(*
IF bToken THEN
	gUI.TiG.arrPV[1].sColumn[3].bExtend		:=arrExecute[20,0];	//E00L
	gUI.TiG.arrPV[1].sColumn[3].bRetract	:=arrExecute[20,1];	
	gUI.TiG.arrPV[1].sColumn[6].bExtend		:=arrExecute[20,2];	//E01L
	gUI.TiG.arrPV[1].sColumn[6].bRetract	:=arrExecute[20,3];	
	gUI.TiG.arrPV[2].sColumn[1].bExtend		:=arrExecute[20,4];	//E02L
	gUI.TiG.arrPV[2].sColumn[1].bRetract	:=arrExecute[20,5];	
	gUI.TiG.arrPV[2].sColumn[2].bExtend		:=arrExecute[20,6];	//E05L
	gUI.TiG.arrPV[2].sColumn[2].bRetract	:=arrExecute[20,7];	
	gUI.TiG.arrPV[2].sColumn[3].bExtend		:=arrExecute[20,8];	//E06L
	gUI.TiG.arrPV[2].sColumn[3].bRetract	:=arrExecute[20,9];	
	gUI.TiG.arrPV[2].sColumn[4].bExtend		:=arrExecute[20,10];//E09L
	gUI.TiG.arrPV[2].sColumn[4].bRetract	:=arrExecute[20,11];	
	gUI.TiG.arrPV[2].sColumn[5].bExtend		:=arrExecute[20,12];//E10L
	gUI.TiG.arrPV[2].sColumn[5].bRetract	:=arrExecute[20,13];	
	gUI.TiG.arrPV[6].sColumn[4].bExtend		:=arrExecute[20,14];//E13L
	gUI.TiG.arrPV[6].sColumn[4].bRetract	:=arrExecute[20,15];	
			
	gUI.TiG.arrPV[6].sColumn[3].bExtend		:=arrExecute[21,0];	//E14L
	gUI.TiG.arrPV[6].sColumn[3].bRetract	:=arrExecute[21,1];	
	gUI.TiG.arrPV[6].sColumn[5].bExtend		:=arrExecute[21,2];	//E16L1
	gUI.TiG.arrPV[6].sColumn[5].bRetract	:=arrExecute[21,3];	
	gUI.TiG.arrPV[7].sColumn[6].bExtend		:=arrExecute[21,4];	//E17L1
	gUI.TiG.arrPV[7].sColumn[6].bRetract	:=arrExecute[21,5];	
	gUI.TiG.arrPV[7].sColumn[1].bExtend		:=arrExecute[21,6];	//E18L
	gUI.TiG.arrPV[7].sColumn[1].bRetract	:=arrExecute[21,7];	
	gUI.TiG.arrPV[7].sColumn[2].bExtend		:=arrExecute[21,8];	//E22L
	gUI.TiG.arrPV[7].sColumn[2].bRetract	:=arrExecute[21,9];	
	gUI.TiG.arrPV[7].sColumn[3].bExtend		:=arrExecute[21,10];//E23L
	gUI.TiG.arrPV[7].sColumn[3].bRetract	:=arrExecute[21,11];	
	gUI.TiG.arrPV[7].sColumn[7].bExtend		:=arrExecute[21,12];//E27L1
	gUI.TiG.arrPV[7].sColumn[7].bRetract	:=arrExecute[21,13];	
	gUI.TiG.arrPV[1].sColumn[1].bExtend		:=arrExecute[21,14];//E28L1
	gUI.TiG.arrPV[1].sColumn[1].bRetract	:=arrExecute[21,15];	
			
	gUI.TiG.arrPV[1].sColumn[2].bExtend		:=arrExecute[22,0];	//E29L
	gUI.TiG.arrPV[1].sColumn[2].bRetract	:=arrExecute[22,1];	
	gUI.TiG.arrPV[3].sColumn[1].bExtend		:=arrExecute[22,2];	//E01Q1
	gUI.TiG.arrPV[3].sColumn[1].bRetract	:=arrExecute[22,3];	
	gUI.TiG.arrPV[4].sColumn[1].bExtend		:=arrExecute[22,4];	//E05Q1
	gUI.TiG.arrPV[4].sColumn[1].bRetract	:=arrExecute[22,5];	
	gUI.TiG.arrPV[5].sColumn[1].bExtend		:=arrExecute[22,6];	//E09Q1
	gUI.TiG.arrPV[5].sColumn[1].bRetract	:=arrExecute[22,7];	
	gUI.TiG.arrPV[6].sColumn[1].bExtend		:=arrExecute[22,8];	//E13Q
	gUI.TiG.arrPV[6].sColumn[1].bRetract	:=arrExecute[22,9];	
	gUI.TiG.arrPV[6].sColumn[2].bExtend		:=arrExecute[22,10];//E15Q
	gUI.TiG.arrPV[6].sColumn[2].bRetract	:=arrExecute[22,11];	
	gUI.TiG.arrPV[7].sColumn[4].bExtend		:=arrExecute[22,12];//E17Q
	gUI.TiG.arrPV[7].sColumn[4].bRetract	:=arrExecute[22,13];	
	gUI.TiG.arrPV[7].sColumn[5].bExtend		:=arrExecute[22,14];//E22Q
	gUI.TiG.arrPV[7].sColumn[5].bRetract	:=arrExecute[22,15];	
			
	gUI.TiG.arrPV[1].sColumn[5].bExtend		:=arrExecute[23,0];//E28Q
	gUI.TiG.arrPV[1].sColumn[5].bRetract	:=arrExecute[23,1];	
	gUI.TiG.arrPV[1].sColumn[4].bExtend		:=arrExecute[23,2];//E29Q
	gUI.TiG.arrPV[1].sColumn[4].bRetract	:=arrExecute[23,3];	

END_IF

IF bToken THEN
	FOR iTemp1:=20 TO 23 DO
	FOR iTemp2:=0 TO 15 DO
		IF arrExecute[iTemp1,iTemp2] AND isArrived(iTemp1,iTemp2) THEN
			arrExecute[iTemp1,iTemp2]:=0;
		END_IF
	END_FOR		
	END_FOR
END_IF
bToken:=FALSE;
*)
END_METHOD

END_PROGRAM

// Device/Application/public_datum/otherContent/modbusold/isArrived
FUNCTION isArrived : BOOL
VAR_INPUT
	i1		:USINT;
	i2		:USINT;
END_VAR
VAR
	iVT		:USINT;
	iVT1	:USINT;
	i2H	:USINT;	//i2Half
	bFetch	:BOOL;
	
END_VAR
VAR CONSTANT
	a0PV		:ARRAY [0..7] OF USINT :=[1,1,2,2,2,2,2,6];	
	a0PV1		:ARRAY [0..7] OF USINT :=[3,6,1,2,3,4,5,4];		
	a1PV		:ARRAY [0..7] OF USINT :=[6,6,7,7,7,7,7,1];	
	a1PV1		:ARRAY [0..7] OF USINT :=[3,5,6,1,2,3,7,1];	
	a2PV		:ARRAY [0..7] OF USINT :=[1,3,4,5,6,6,7,7];	
	a2PV1		:ARRAY [0..7] OF USINT :=[2,1,1,1,1,2,4,5];		
	a3PV		:ARRAY [0..7] OF USINT :=[1,1];	
	a3PV1		:ARRAY [0..7] OF USINT :=[5,4];	
END_VAR

bFetch:=FALSE;
i2H:=i2/2;
IF i2 MOD 2 =0 THEN//伸出指令
	CASE i1 OF
	20:
		IF gImple.PV_GroupTi.arrPV[a0PV[i2H]].sColumn[a0PV1[i2H]].eStat=cmdStat.Extend_Done THEN
			bFetch:=TRUE;
		END_IF
	21:
		IF gImple.PV_GroupTi.arrPV[a1PV[i2H]].sColumn[a1PV1[i2H]].eStat=cmdStat.Extend_Done THEN
			bFetch:=TRUE;
		END_IF		
	22:
		IF gImple.PV_GroupTi.arrPV[a2PV[i2H]].sColumn[a2PV1[i2H]].eStat=cmdStat.Extend_Done THEN
			bFetch:=TRUE;
		END_IF		
	23:
		IF gImple.PV_GroupTi.arrPV[a2PV[i2H]].sColumn[a2PV1[i2H]].eStat=cmdStat.Extend_Done THEN
			bFetch:=TRUE;
		END_IF		
	END_CASE
ELSE				//缩回指令
		CASE i1 OF
	20:
		IF gImple.PV_GroupTi.arrPV[a0PV[i2H]].sColumn[a0PV1[i2H]].eStat=cmdStat.Retract_Done THEN
			bFetch:=TRUE;
		END_IF
	21:
		IF gImple.PV_GroupTi.arrPV[a1PV[i2H]].sColumn[a1PV1[i2H]].eStat=cmdStat.Retract_Done THEN
			bFetch:=TRUE;
		END_IF		
	22:
		IF gImple.PV_GroupTi.arrPV[a2PV[i2H]].sColumn[a2PV1[i2H]].eStat=cmdStat.Retract_Done THEN
			bFetch:=TRUE;
		END_IF		
	23:
		IF gImple.PV_GroupTi.arrPV[a2PV[i2H]].sColumn[a2PV1[i2H]].eStat=cmdStat.Retract_Done THEN
			bFetch:=TRUE;
		END_IF		
	END_CASE
END_IF


isArrived:=bFetch;

END_FUNCTION

// Device/Application/public_datum/otherContent/rail_rotate/rotatePlatAct
PROGRAM rotatePlatAct
VAR
		bInitialize		:BOOL:=TRUE;
		iTemp			:INT;
		//fbPercentCalc	:percentCalc;
		iV1:INT;
		iV2:INT;
END_VAR

(*
IF bInitialize THEN	//初始化
	rotatePlatAct.initParam();
END_IF
rotatePlatAct.statusDisplayA();
rotatePlatAct.commandDeliverDi();
*)
IF gImple.PV_GroupTi.arrRotSYN.sStatus.oilExtend_Done THEN
	gImple.PV_GroupTi.arrRotSYN.sStatus.oilStat:=cmdStat.Extend_Done;
	gUI.TiG.sRotLed.oilExtended:=TRUE;gUI.TiG.sRotLed.oilRetracted:=FALSE;
END_IF
IF gImple.PV_GroupTi.arrRotSYN.sStatus.oilRetract_Done THEN
	gImple.PV_GroupTi.arrRotSYN.sStatus.oilStat:=cmdStat.Retract_Done;
	gUI.TiG.sRotLed.oilExtended:=FALSE;gUI.TiG.sRotLed.oilRetracted:=TRUE;
END_IF
IF gImple.PV_GroupTi.arrRotSYN.sStatus.rotFront_Done THEN
	gImple.PV_GroupTi.arrRotSYN.sStatus.rotplatformStat:=cmdStat.Extend_Done;
	gUI.TiG.sRotLed.platExtended:=TRUE;gUI.TiG.sRotLed.platRetracted:=FALSE;
END_IF
IF gImple.PV_GroupTi.arrRotSYN.sStatus.rotReverse_Done THEN
	gImple.PV_GroupTi.arrRotSYN.sStatus.rotplatformStat:=cmdStat.Retract_Done;
	gUI.TiG.sRotLed.platExtended:=FALSE;gUI.TiG.sRotLed.platRetracted:=TRUE;
END_IF


	IF gUI.TiG.sRot.oilExtend  THEN
		IF gImple.PV_GroupTi.arrRotSYN.sStatus.oilStat=cmdStat.Extend_Done THEN
			//gImple.PV_GroupTi.arrRotSYN.sStatus.oilCnt:=0;
			gUI.TiG.sRot.oilExtend:=FALSE;
			gImple.PV_GroupTi.arrRotSYN.sCtrl.oilExtend:=FALSE;			
		ELSE
			gImple.PV_GroupTi.arrRotSYN.sStatus.oilStat:=cmdStat.eRun;
			gImple.PV_GroupTi.arrRotSYN.sCtrl.oilExtend:=TRUE;
			gImple.PV_GroupTi.arrRotSYN.sCtrl.oilRetract:=FALSE;
			gUI.TiG.sRot.oilRetract:=FALSE;
		END_IF
	ELSE
		gImple.PV_GroupTi.arrRotSYN.sCtrl.oilExtend:=FALSE;
	END_IF
	
	IF gUI.TiG.sRot.oilRetract  THEN
		IF gImple.PV_GroupTi.arrRotSYN.sStatus.oilStat=cmdStat.Retract_Done THEN
			//gImple.PV_GroupTi.arrRotSYN.sStatus.oilCnt:=0;
			gUI.TiG.sRot.oilRetract:=FALSE;
			gImple.PV_GroupTi.arrRotSYN.sCtrl.oilRetract:=FALSE;
		ELSE
			gImple.PV_GroupTi.arrRotSYN.sStatus.oilStat:=cmdStat.eRun;
			gImple.PV_GroupTi.arrRotSYN.sCtrl.oilRetract:=TRUE;
			gImple.PV_GroupTi.arrRotSYN.sCtrl.oilExtend:=FALSE;	
			gUI.TiG.sRot.oilExtend:=FALSE;	
		END_IF
	ELSE
		gImple.PV_GroupTi.arrRotSYN.sCtrl.oilRetract:=FALSE;
	END_IF	




	IF gUI.TiG.sRot.rotFront  THEN
		IF gImple.PV_GroupTi.arrRotSYN.sStatus.rotplatformStat=cmdStat.Extend_Done THEN
			gUI.TiG.sRot.rotFront:=FALSE;
			gImple.PV_GroupTi.arrRotSYN.sCtrl.rotFront:=FALSE;			
		ELSE 
			gImple.PV_GroupTi.arrRotSYN.sStatus.rotplatformStat:=cmdStat.eRun;
			gImple.PV_GroupTi.arrRotSYN.sCtrl.rotFront:=TRUE;
			gImple.PV_GroupTi.arrRotSYN.sCtrl.rotReverse:=FALSE;	
			gUI.TiG.sRot.rotReverse:=FALSE;
		END_IF
	ELSE
		gImple.PV_GroupTi.arrRotSYN.sCtrl.rotFront:=FALSE;
	END_IF
	
	IF gUI.TiG.sRot.rotReverse  THEN
		IF gImple.PV_GroupTi.arrRotSYN.sStatus.rotplatformStat=cmdStat.Retract_Done THEN
			gUI.TiG.sRot.rotReverse:=FALSE;
			gImple.PV_GroupTi.arrRotSYN.sCtrl.rotReverse:=FALSE;	
		ELSE
			gImple.PV_GroupTi.arrRotSYN.sStatus.rotplatformStat:=cmdStat.eRun;
			gImple.PV_GroupTi.arrRotSYN.sCtrl.rotReverse:=TRUE;
			gImple.PV_GroupTi.arrRotSYN.sCtrl.rotFront:=FALSE;	
			gUI.TiG.sRot.rotFront:=FALSE;
		END_IF
	ELSE
		gImple.PV_GroupTi.arrRotSYN.sCtrl.rotReverse:=FALSE;	
	END_IF

ACTION initParam:
gUI.DiG.arrSYN[31].sNum[1].strName:='D31Q';
gUI.DiG.arrSYN[31].sNum[2].strName:='D31Q1';
gUI.DiG.arrSYN[31].sNum[3].strName:='D31Q2';

gUI.DiG.arrSYN[32].sNum[1].strName:='D32Q';
gUI.DiG.arrSYN[32].sNum[2].strName:='D32Q1';
gUI.DiG.arrSYN[32].sNum[3].strName:='D32Q2';


gUI.TiG.arrSYN[31].sNum[1].strName:='E31Q';
gUI.TiG.arrSYN[31].sNum[2].strName:='E31Q1';
gUI.TiG.arrSYN[32].sNum[1].strName:='E32Q';
gUI.TiG.arrSYN[32].sNum[2].strName:='E32Q2';


//gImple.PV_GroupDi.arrRotSYN[31].arrNum[1].posVal.Retract:=2;
//gImple.PV_GroupDi.arrRotSYN[31].arrNum[1].posVal.Extend:=200;
END_ACTION

ACTION statusDisplayA:
gUI.DiG.arrSYN[31].sNum[1].rPosition:=gImple.PV_GroupDi.arrRotSYN[31].sNum[1].posVal.Current;
gUI.DiG.arrSYN[31].sNum[2].rPosition:=gImple.PV_GroupDi.arrRotSYN[31].sNum[2].posVal.Current;
gUI.DiG.arrSYN[31].sNum[3].rPosition:=gImple.PV_GroupDi.arrRotSYN[31].sNum[3].posVal.Current;

gUI.TiG.arrSYN[31].sNum[1].rPosition:=gImple.PV_GroupTi.arrRotSYN[31].sNum[1].posVal.Current;
gUI.TiG.arrSYN[31].sNum[2].rPosition:=gImple.PV_GroupTi.arrRotSYN[31].sNum[2].posVal.Current;

FOR iTemp:=1 TO 3 DO
	fbPercentCalc(rInput:=gImple.PV_GroupDi.arrRotSYN[31].sNum[iTemp].posVal.Current,
			rExtend:=gImple.PV_GroupDi.arrRotSYN[31].sNum[iTemp].posVal.Extend,
			rRetract:=gImple.PV_GroupDi.arrRotSYN[31].sNum[iTemp].posVal.Retract,
			rOut=>);
	gUI.DiG.arrSYN[31].sNum[iTemp].rPercent:=fbPercentCalc.rOut;
	fbPercentCalc(rInput:=gImple.PV_GroupDi.arrRotSYN[32].sNum[iTemp].posVal.Current,
			rExtend:=gImple.PV_GroupDi.arrRotSYN[32].sNum[iTemp].posVal.Extend,
			rRetract:=gImple.PV_GroupDi.arrRotSYN[32].sNum[iTemp].posVal.Retract,
			rOut=>);
	gUI.DiG.arrSYN[32].sNum[iTemp].rPercent:=fbPercentCalc.rOut;
END_FOR

FOR iTemp:=1 TO 2 DO
	fbPercentCalc(rInput:=gImple.PV_GroupTi.arrRotSYN[31].sNum[iTemp].posVal.Current,
			rExtend:=gImple.PV_GroupTi.arrRotSYN[31].sNum[iTemp].posVal.Extend,
			rRetract:=gImple.PV_GroupTi.arrRotSYN[31].sNum[iTemp].posVal.Retract,
			rOut=>);
	gUI.TiG.arrSYN[31].sNum[iTemp].rPercent:=fbPercentCalc.rOut;
	fbPercentCalc(rInput:=gImple.PV_GroupTi.arrRotSYN[32].sNum[iTemp].posVal.Current,
			rExtend:=gImple.PV_GroupTi.arrRotSYN[32].sNum[iTemp].posVal.Extend,
			rRetract:=gImple.PV_GroupTi.arrRotSYN[32].sNum[iTemp].posVal.Retract,
			rOut=>);
	gUI.TiG.arrSYN[32].sNum[iTemp].rPercent:=fbPercentCalc.rOut;	
END_FOR
END_ACTION

METHOD PRIVATE commandDeliverDi : BOOL
VAR_INPUT
END_VAR
VAR
		eCommand				:cmdStat;
		iCount					:UINT;	
		iCntErr					:UINT:=200*15;			//超时时间15s
		eUnitIndex				:INT;
		fbCheckGroup				:ARRAY[31..32,1..2] OF syncUnitCheck;
		arrOBUSP				:ARRAY[1..2] OF OilBlockUnit_Status_PosVal;

END_VAR
FOR iV1:=31 TO 32 DO
	FOR iV2:=1 TO 2 DO
		iCount:=gImple.PV_GroupDi.arrRotSYN[iV1].iCntErr[iV2];
		IF gUI.DiG.arrSYN[iV1].sColumn[iV2].bExtend<>gUI.DiG.arrSYN[iV1].sColumn[iV2].bRetract THEN
			gImple.PV_GroupDi.arrRotSYN[iV1].sColumn[iV2].eStat:=cmdStat.eRun;
			IF gUI.DiG.arrSYN[iV1].sColumn[iV2].bExtend THEN
				eCommand:=cmdStat.cExtend;
			END_IF
			IF gUI.DiG.arrSYN[iV1].sColumn[iV2].bRetract THEN
				eCommand:=cmdStat.cRetract;
			END_IF
		ELSE	
			eCommand:=cmdStat.cStop;
		END_IF
		IF gUI.DiG.arrSYN[iV1].sColumn[iV2].bStop THEN
			eCommand:=cmdStat.cStop;
		END_IF
		
		arrOBUSP[1].Current:=gImple.PV_GroupDi.arrRotSYN[iV1].sNum[iV2].posVal.Current;
		arrOBUSP[1].Extend:=gImple.PV_GroupDi.arrRotSYN[iV1].sNum[iV2].posVal.Extend;
		arrOBUSP[1].Retract:=gImple.PV_GroupDi.arrRotSYN[iV1].sNum[iV2].posVal.Retract;
		IF iV2=2 THEN
			arrOBUSP[2].Current:=gImple.PV_GroupDi.arrRotSYN[iV1].sNum[iV2].posVal.Current;
			arrOBUSP[2].Extend:=gImple.PV_GroupDi.arrRotSYN[iV1].sNum[iV2].posVal.Extend;
			arrOBUSP[2].Retract:=gImple.PV_GroupDi.arrRotSYN[iV1].sNum[iV2].posVal.Retract;
		ELSE
			arrOBUSP[2].Current:=0;	arrOBUSP[2].Extend:=0;arrOBUSP[2].Retract:=0;
		END_IF
		
		fbCheckGroup[iV1,iV2](
			arrPosVal:=arrOBUSP,
			cmdAct:=eCommand,
			bFetch	=>);
		
		IF fbCheckGroup[iV1,iV2].bFetch=TRUE THEN
			iCount:=0;
			IF gImple.PV_GroupDi.arrRotSYN[iV1].sColumn[iV2].eStat<>cmdStat.eError THEN
				//正常态油缸指令复位
				gUI.DiG.arrSYN[iV1].sColumn[iV2].bStop:=FALSE;
				gUI.DiG.arrSYN[iV1].sColumn[iV2].bExtend:=FALSE;
				gUI.DiG.arrSYN[iV1].sColumn[iV2].bRetract:=FALSE;	
				//SyncCmdExecuteD(ADR(gImple.PV_GroupTi),iV1,iV2,cmdStat.cStop);
				//判断每个开关阀的总状态（伸出or收回）	
				fbCheckGroup[iV1,iV2](cmdAct:=cmdStat.cExtend,arrPosVal:=arrOBUSP);
				IF fbCheckGroup[iV1,iV2].bFetch=TRUE THEN
					gImple.PV_GroupDi.arrRotSYN[iV1].sColumn[iV2].eStat:=cmdStat.Extend_Done;
				END_IF
				fbCheckGroup[iV1,iV2](cmdAct:=cmdStat.cRetract,arrPosVal:=arrOBUSP);
				IF fbCheckGroup[iV1,iV2].bFetch=TRUE THEN
					gImple.PV_GroupDi.arrRotSYN[iV1].sColumn[iV2].eStat:=cmdStat.Retract_Done;
				END_IF			
				//都不是则为Normal态
				IF gImple.PV_GroupDi.arrRotSYN[iV1].sColumn[iV2].eStat<>cmdStat.Retract_Done AND gImple.PV_GroupDi.arrRotSYN[iV1].sColumn[iV2].eStat<>cmdStat.Extend_Done THEN
					gImple.PV_GroupDi.arrRotSYN[iV1].sColumn[iV2].eStat:=cmdStat.eNormal;
				END_IF
				
			END_IF
		ELSE
			iCount:= iCount +1;
			gImple.PV_GroupDi.arrRotSYN[iV1].sColumn[iV2].eStat:=cmdStat.eRun;
			//SyncCmdExecuteD(ADR(gImple.PV_GroupTi),iV1,iV2,eCommand);
		END_IF
		
		IF iCount>=iCntErr THEN
			//错误态油缸指令复位
			gImple.PV_GroupDi.arrRotSYN[iV1].sColumn[iV2].eStat:=cmdStat.eError;
			gUI.DiG.arrSYN[iV1].sColumn[iV2].bStop:=FALSE;
			gUI.DiG.arrSYN[iV1].sColumn[iV2].bExtend:=FALSE;
			gUI.DiG.arrSYN[iV1].sColumn[iV2].bRetract:=FALSE;	
			//SyncCmdExecuteD(ADR(gImple.PV_GroupTi),iV1,iV2,cmdStat.cStop);
		END_IF		
		gImple.PV_GroupDi.arrRotSYN[iV1].iCntErr[iV2]:=iCount;
	END_FOR
END_FOR
END_METHOD

METHOD PRIVATE commandDeliverTi : BOOL
VAR_INPUT
END_VAR
VAR
		eCommand				:cmdStat;
		iCount					:UINT;	
		iCntErr					:UINT:=200*15;			//超时时间15s
		eUnitIndex				:INT;
		fbCheckGroup				:ARRAY[31..32,1..2] OF syncUnitCheck;
		arrOBUSP				:ARRAY[1..2] OF OilBlockUnit_Status_PosVal;

END_VAR
FOR iV1:=31 TO 32 DO
	FOR iV2:=1 TO 2 DO
		iCount:=gImple.PV_GroupTi.arrRotSYN[iV1].iCntErr[iV2];
		IF gUI.TiG.arrSYN[iV1].sColumn[iV2].bExtend<>gUI.TiG.arrSYN[iV1].sColumn[iV2].bRetract THEN
			gImple.PV_GroupTi.arrRotSYN[iV1].sColumn[iV2].eStat:=cmdStat.eRun;
			IF gUI.TiG.arrSYN[iV1].sColumn[iV2].bExtend THEN
				eCommand:=cmdStat.cExtend;
			END_IF
			IF gUI.TiG.arrSYN[iV1].sColumn[iV2].bRetract THEN
				eCommand:=cmdStat.cRetract;
			END_IF
		ELSE	
			eCommand:=cmdStat.cStop;
		END_IF
		IF gUI.TiG.arrSYN[iV1].sColumn[iV2].bStop THEN
			eCommand:=cmdStat.cStop;
		END_IF
		
		arrOBUSP[1].Current:=gImple.PV_GroupTi.arrRotSYN[iV1].sNum[iV2].posVal.Current;
		arrOBUSP[1].Extend:=gImple.PV_GroupTi.arrRotSYN[iV1].sNum[iV2].posVal.Extend;
		arrOBUSP[1].Retract:=gImple.PV_GroupTi.arrRotSYN[iV1].sNum[iV2].posVal.Retract;
		arrOBUSP[2].Current:=0;	arrOBUSP[2].Extend:=0;arrOBUSP[2].Retract:=0;

		
		fbCheckGroup[iV1,iV2](
			arrPosVal:=arrOBUSP,
			cmdAct:=eCommand,
			bFetch	=>);
		
		IF fbCheckGroup[iV1,iV2].bFetch=TRUE THEN
			iCount:=0;
			IF gImple.PV_GroupTi.arrRotSYN[iV1].sColumn[iV2].eStat<>cmdStat.eError THEN
				//正常态油缸指令复位
				gUI.TiG.arrSYN[iV1].sColumn[iV2].bStop:=FALSE;
				gUI.TiG.arrSYN[iV1].sColumn[iV2].bExtend:=FALSE;
				gUI.TiG.arrSYN[iV1].sColumn[iV2].bRetract:=FALSE;	
				//SyncCmdExecuteT(ADR(gImple.PV_GroupTi),iV1,iV2,cmdStat.cStop);
				//判断每个开关阀的总状态（伸出or收回）	
				fbCheckGroup[iV1,iV2](cmdAct:=cmdStat.cExtend,arrPosVal:=arrOBUSP);
				IF fbCheckGroup[iV1,iV2].bFetch=TRUE THEN
					gImple.PV_GroupTi.arrRotSYN[iV1].sColumn[iV2].eStat:=cmdStat.Extend_Done;
				END_IF
				fbCheckGroup[iV1,iV2](cmdAct:=cmdStat.cRetract,arrPosVal:=arrOBUSP);
				IF fbCheckGroup[iV1,iV2].bFetch=TRUE THEN
					gImple.PV_GroupTi.arrRotSYN[iV1].sColumn[iV2].eStat:=cmdStat.Retract_Done;
				END_IF			
				//都不是则为Normal态
				IF gImple.PV_GroupTi.arrRotSYN[iV1].sColumn[iV2].eStat<>cmdStat.Retract_Done AND gImple.PV_GroupTi.arrRotSYN[iV1].sColumn[iV2].eStat<>cmdStat.Extend_Done THEN
					gImple.PV_GroupTi.arrRotSYN[iV1].sColumn[iV2].eStat:=cmdStat.eNormal;
				END_IF
				
			END_IF
		ELSE
			iCount:= iCount +1;
			gImple.PV_GroupTi.arrRotSYN[iV1].sColumn[iV2].eStat:=cmdStat.eRun;
			//SyncCmdExecuteT(ADR(gImple.PV_GroupTi),iV1,iV2,eCommand);
		END_IF
		
		IF iCount>=iCntErr THEN
			//错误态油缸指令复位
			gImple.PV_GroupTi.arrRotSYN[iV1].sColumn[iV2].eStat:=cmdStat.eError;
			gUI.TiG.arrSYN[iV1].sColumn[iV2].bStop:=FALSE;
			gUI.TiG.arrSYN[iV1].sColumn[iV2].bExtend:=FALSE;
			gUI.TiG.arrSYN[iV1].sColumn[iV2].bRetract:=FALSE;	
			//SyncCmdExecuteT(ADR(gImple.PV_GroupTi),iV1,iV2,cmdStat.cStop);
		END_IF		
		gImple.PV_GroupTi.arrRotSYN[iV1].iCntErr[iV2]:=iCount;
	END_FOR
END_FOR
END_METHOD

END_PROGRAM

// Device/Application/public_datum/cmdcheck/syncUnitCheck
FUNCTION_BLOCK syncUnitCheck
VAR_INPUT
	arrPosVal	:ARRAY  [1..2] OF OilBlockUnit_Status_PosVal;

	cmdAct		:cmdStat;
	
END_VAR
VAR_OUTPUT
	bFetch		:BOOL;
END_VAR
VAR
	iCheck			:INT;
	iNum			:INT;				//有值的位移传感器值
	outStat			:ARRAY[1..2] OF OilBlockUnit_Status_Loc;
	iTemp			:INT;
	bAllDone		:BOOL;
END_VAR

iNum:=0;
FOR iTemp :=1 TO 2 DO
	IF arrPosVal[iTemp].Extend <> 0 THEN
		iNum:=iNum+1;
	END_IF
END_FOR
FOR iCheck:=1 TO iNum DO
	outStat[iCheck]	:=fGetUnitStat(arrPosVal[iCheck].Extend,arrPosVal[iCheck].Retract,arrPosVal[iCheck].Current,2.0);
END_FOR


bAllDone:=TRUE;

	//有一个未到指令位置则未完成
	CASE cmdAct OF 
		cmdStat.cExtend:
			FOR iCheck:=1 TO iNum DO
				IF outStat[iCheck]<>OilBlockUnit_Status_Loc.eExtended THEN
					bAllDone:=FALSE;
				END_IF
			END_FOR
		cmdStat.cRetract:
			FOR iCheck:=1 TO iNum DO
				IF outStat[iCheck]<>OilBlockUnit_Status_Loc.eRetracted THEN
					bAllDone:=FALSE;
				END_IF
			END_FOR	
		cmdStat.cStop:
			
	END_CASE

IF bAllDone THEN
	bFetch	:= TRUE;
ELSE
	bFetch	:= FALSE;
END_IF

END_FUNCTION_BLOCK

// Device/Application/can/swmc_floor_rail/swmc_C03_Rx
FUNCTION swmc_C03_Rx : BOOL
VAR_INPUT
	CNT				: UINT;
	//psPVDi			: POINTER TO propValveModule_Di;
	psPVTi			: POINTER TO propValveModule_Ti;
END_VAR
VAR
	frame	 	    : Can_baseframe;
	COB_ID			: UINT;
	I				: UINT;
	pos				: WORD;
END_VAR

IF gCan.C3RxMsg.RxCounter <>  gCan.C3RxCounter THEN    //接收到新的数据

	FOR  I := 1 TO  gCan.C3RxMsg.NoOfRxMessages DO
		frame :=CAN_Read_Data_SWMC(3,I);
		COB_ID :=	frame.id;    //获取ID
		CASE COB_ID OF     //根据ID解析协议
	
			//C3-0x330
			16#330:           //接收C3送来的数据

				psPVTi^.arrRotSYN.sStatus.oilExtend_Done := frame.data[1].0;
				psPVTi^.arrRotSYN.sStatus.oilRetract_Done:= frame.data[1].1;
				
				psPVTi^.arrRotSYN.sStatus.rotFront_Done  := frame.data[2].0;
				psPVTi^.arrRotSYN.sStatus.rotReverse_Done:= frame.data[2].1;
				
		END_CASE
	END_FOR


	gCan.C3RxCounter := gCan.C3RxMsg.RxCounter ;
END_IF

END_FUNCTION

// Device/Application/can/swmc_floor_rail/swmc_C03_Tx
FUNCTION swmc_C03_Tx : BOOL
VAR_INPUT
	CNT				: UINT;
	
	//psPVDi			: POINTER TO propValveModule_Di;
	psPVTi			: POINTER TO propValveModule_Ti;

END_VAR
VAR
	senddata	: ARRAY[1..8] OF BYTE;
	Send_cnt	: UINT;
END_VAR

//速度控制--待定
Send_cnt :=  CNT MOD 3;

CASE Send_cnt OF
	
	1:
 	//C3-0x430
	senddata[1].0 := psPVTi^.arrRotSYN.sCtrl.oilExtend;
	senddata[1].1 := psPVTi^.arrRotSYN.sCtrl.oilRetract;
	
	senddata[2].0 := psPVTi^.arrRotSYN.sCtrl.rotFront;
	senddata[2].1 := psPVTi^.arrRotSYN.sCtrl.rotReverse;	

	//发送至C3
	CAN_Send_Data_SWMC(3, 16#430,senddata);				//发送ID 0x430到C3

END_CASE

END_FUNCTION

// Device/Application/display/OrigDi/YY_Station_Display
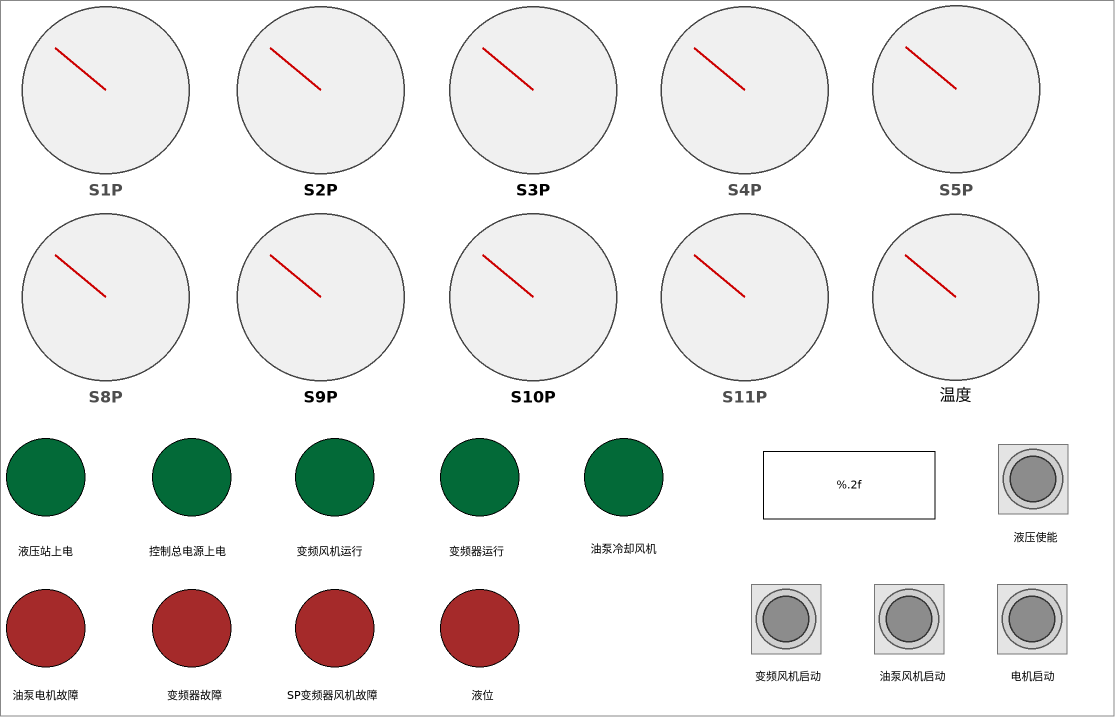
VISUALIZATION YY_Station_Display  // 1115x717
    Ellipse (6,438 79x78), colour toggle: gUI.bYysPower
    Ellipse (152,438 79x78), colour toggle: gUI.bCtrlPower
    Ellipse (295,438 79x78), colour toggle: gUI.bFreqConverterFan
    Ellipse (440,438 79x78), colour toggle: gUI.bFreqConverter
    Label (6,532 79x39), "液压站上电"
    Label (110,532 155x39), "控制总电源上电"
    Label (252,532 155x39), "变频风机运行"
    Label (437,532 79x39), "变频器运行"
    Ellipse (6,589 79x78), colour toggle: gUI.bOilPumpM_Fault
    Ellipse (152,589 79x78), colour toggle: gUI.bFreqConverter_Fault
    Label (6,676 79x39), "油泵电机故障"
    Label (584,532 79x34), "油泵冷却风机"
    Label (117,676 155x39), "变频器故障"
    Ellipse (295,589 79x78), colour toggle: gUI.bFreqConverterFan_Fault
    Label (255,676 155x39), "SP变频器风机故障"
    Ellipse (440,589 79x78), colour toggle: gUI.bFluidLevel
    Label (443,676 79x39), "液位"
    PushSwitchLed (751,584 70x70), variable: gUI.cmdInverterFan, behaviour: TOGGLE, style: Switch-PushSwitchLed-Gray
    PushSwitchLed (874,584 70x70), variable: gUI.cmdOilPumpFan, behaviour: TOGGLE, style: Switch-PushSwitchLed-Gray
    Label (740,657 96x39), "变频风机启动"
    Label (835,657 155x39), "油泵风机启动"
    PushSwitchLed (997,584 70x70), variable: gUI.cmdOilPumpM, behaviour: TOGGLE, style: Switch-PushSwitchLed-Gray
    Label (955,657 155x39), "电机启动"
    Rectangle (763,451 172x68), "%.2f", text variable: gUI.cmdOilPrePercent
        OnMouseDown: write the text variable via Default, min 0, max 100
    Label (958,518 155x39), "液压使能"
    PushSwitchLed (998,444 70x70), variable: gUI.cmdOilPre_EN, behaviour: TOGGLE, style: Switch-PushSwitchLed-Gray
    Ellipse (584,438 79x78), colour toggle: gUI.bOilPumpFan
    Meter360 (872,5 168x168), value: gUI.arrStationPressure[5], style: Meter-Meter360-Gray, scale format: %.1f, scale 0..200
        p518627256: bar
    Label (872,175 168x30), "S5P"
    Meter360 (872,213 167x168), value: gUI.rTemperature, style: Meter-Meter360-Gray, scale format: %.1f, scale 0..200
        p518627256: bar
    Label (872,380 167x30), "温度"
    Meter360 (18,6 175x168), value: gUI.arrStationPressure[1], style: Meter-Meter360-Gray, scale format: %.1f, scale 0..100
        p518627256: bar
    Label (18,175 175x30), "S1P"
    Meter360 (18,213 175x168), value: gUI.arrStationPressure[8], style: Meter-Meter360-Gray, scale format: %.1f, scale 0..100
        p518627256: bar
    Label (18,382 175x30), "S8P"
    Meter360 (234,6 173x168), value: gUI.arrStationPressure[2], style: Meter-Meter360-Gray, scale format: %.1f, scale 0..100
        p518627256: bar
    Label (234,175 173x30), "S2P"
    Meter360 (234,213 173x168), value: gUI.arrStationPressure[9], style: Meter-Meter360-Gray, scale format: %.1f, scale 0..100
        p518627256: bar
    Label (234,382 173x30), "S9P"
    Meter360 (448,6 170x168), value: gUI.arrStationPressure[3], style: Meter-Meter360-Gray, scale format: %.1f, scale 0..100
        p518627256: bar
    Label (448,175 170x30), "S3P"
    Meter360 (448,213 170x168), value: gUI.arrStationPressure[10], style: Meter-Meter360-Gray, scale format: %.1f, scale 0..100
        p518627256: bar
    Label (448,382 170x30), "S10P"
    Meter360 (659,6 171x168), value: gUI.arrStationPressure[4], style: Meter-Meter360-Gray, scale format: %.1f, scale 0..100
        p518627256: bar
    Label (659,175 171x30), "S4P"
    Meter360 (659,213 171x168), value: gUI.arrStationPressure[11], style: Meter-Meter360-Gray, scale format: %.1f, scale 0..100
        p518627256: bar
    Label (659,382 171x30), "S11P"
END_VISUALIZATION

// Device/Application/display/Module/OilBlock_PrimButton
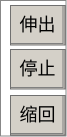
VISUALIZATION OilBlock_PrimButton  // 67x137
VAR_IN_OUT
	extendButton		: BOOL;
	retractButton		: BOOL;
	stopButton			: BOOL;
	
END_VAR
    Button (10,95 55x40), "缩回"
        toggle retractButton
    Button (10,49 55x40), "停止"
        toggle stopButton
    Button (10,5 55x40), "伸出"
        toggle extendButton
END_VISUALIZATION

// Device/Application/display/Module/OilBlock_PrimInfo
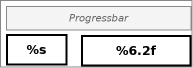
VISUALIZATION OilBlock_PrimInfo  // 193x68
VAR_IN_OUT
	nameStr		:STRING;
	posVal		:REAL;
	percentBar	:REAL;
END_VAR
    RoundedRectangle (6,34 61x31), "%s", text variable: nameStr
    RoundedRectangle (81,35 110x31), "%6.2f", text variable: posVal
    Progressbar (6,6 185x24), variable: percentBar
END_VISUALIZATION

// Device/Application/display/Module/old/Floor_Rail1o
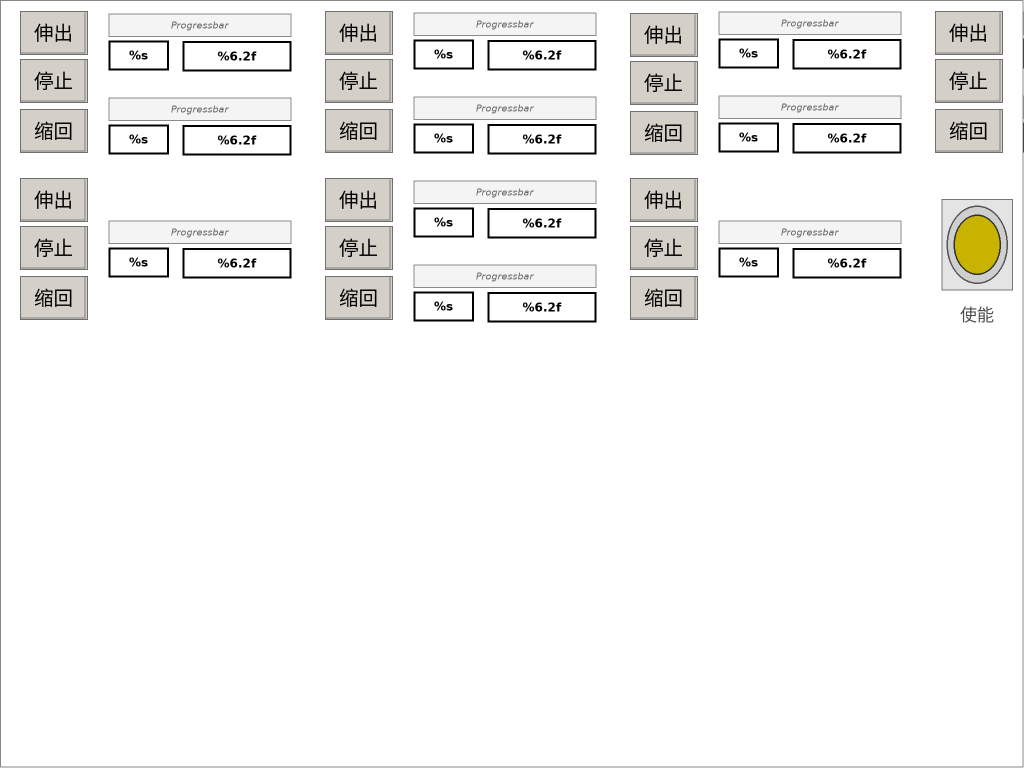
VISUALIZATION Floor_Rail1o  // 1024x768
    Group (8,6 285x151)
        Frame (0,0 82x149)
            shows OilBlock_PrimButton(extendButton := gUI.DiG1.S1.bExtend, retractButton := gUI.DiG1.S1.bRetract, stopButton := gUI.DiG1.S1.bStop)
        Group (95,2 190x149)
            Frame (0,0 190x65)
                shows OilBlock_PrimInfo(nameStr := gUI.DiG1.D00Q1.strName, posVal := gUI.DiG1.D00Q1.rPosition, percentBar := gUI.DiG1.D00Q1.rPercent)
            Frame (0,84 190x65)
                shows OilBlock_PrimInfo(nameStr := gUI.DiG1.D00Q2.strName, posVal := gUI.DiG1.D00Q2.rPosition, percentBar := gUI.DiG1.D00Q2.rPercent)
    Group (313,6 285x150)
        Group (95,1 190x149)
            Frame (0,0 190x65)
                shows OilBlock_PrimInfo(nameStr := gUI.DiG1.D28L1.strName, posVal := gUI.DiG1.D28L1.rPosition, percentBar := gUI.DiG1.D28L1.rPercent)
            Frame (0,84 190x65)
                shows OilBlock_PrimInfo(nameStr := gUI.DiG1.D28L2.strName, posVal := gUI.DiG1.D28L2.rPosition, percentBar := gUI.DiG1.D28L2.rPercent)
        Frame (0,0 82x149)
            shows OilBlock_PrimButton(extendButton := gUI.DiG1.S2.bExtend, retractButton := gUI.DiG1.S2.bRetract, stopButton := gUI.DiG1.S2.bStop)
    Group (618,6 285x151)
        Group (95,0 190x149)
            Frame (0,0 190x65)
                shows OilBlock_PrimInfo(nameStr := gUI.DiG1.D29L.strName, posVal := gUI.DiG1.D29L.rPosition, percentBar := gUI.DiG1.D29L.rPercent)
            Frame (0,84 190x65)
                shows OilBlock_PrimInfo(nameStr := gUI.DiG1.D30L.strName, posVal := gUI.DiG1.D30L.rPosition, percentBar := gUI.DiG1.D30L.rPercent)
        Frame (0,2 82x149)
            shows OilBlock_PrimButton(extendButton := gUI.DiG1.S3.bExtend, retractButton := gUI.DiG1.S3.bRetract, stopButton := gUI.DiG1.S3.bStop)
    Group (923,6 285x149)
        Group (95,0 190x149)
            Frame (0,0 190x65)
                shows OilBlock_PrimInfo(nameStr := gUI.DiG1.D00L1.strName, posVal := gUI.DiG1.D00L1.rPosition, percentBar := gUI.DiG1.D00L1.rPercent)
            Frame (0,84 190x65)
                shows OilBlock_PrimInfo(nameStr := gUI.DiG1.D00L2.strName, posVal := gUI.DiG1.D00L2.rPosition, percentBar := gUI.DiG1.D00L2.rPercent)
        Frame (0,0 82x149)
            shows OilBlock_PrimButton(extendButton := gUI.DiG1.S4.bExtend, retractButton := gUI.DiG1.S4.bRetract, stopButton := gUI.DiG1.S4.bStop)
    Frame (103,215 190x65)
        shows OilBlock_PrimInfo(nameStr := gUI.DiG1.D01L.strName, posVal := gUI.DiG1.D01L.rPosition, percentBar := gUI.DiG1.D01L.rPercent)
    Frame (8,173 82x149)
        shows OilBlock_PrimButton(extendButton := gUI.DiG1.S5.bExtend, retractButton := gUI.DiG1.S5.bRetract, stopButton := gUI.DiG1.S5.bStop)
    Group (313,173 285x151)
        Group (95,2 190x149)
            Frame (0,0 190x65)
                shows OilBlock_PrimInfo(nameStr := gUI.DiG1.D28Q.strName, posVal := gUI.DiG1.D28Q.rPosition, percentBar := gUI.DiG1.D28Q.rPercent)
            Frame (0,84 190x65)
                shows OilBlock_PrimInfo(nameStr := gUI.DiG1.D29Q.strName, posVal := gUI.DiG1.D29Q.rPosition, percentBar := gUI.DiG1.D29Q.rPercent)
        Frame (0,0 82x149)
            shows OilBlock_PrimButton(extendButton := gUI.DiG1.S6.bExtend, retractButton := gUI.DiG1.S6.bRetract, stopButton := gUI.DiG1.S6.bStop)
    Group (618,173 285x149)
        Frame (95,42 190x65)
            shows OilBlock_PrimInfo(nameStr := gUI.DiG1.D30Q.strName, posVal := gUI.DiG1.D30Q.rPosition, percentBar := gUI.DiG1.D30Q.rPercent)
        Frame (0,0 82x149)
            shows OilBlock_PrimButton(extendButton := gUI.DiG1.S7.bExtend, retractButton := gUI.DiG1.S7.bRetract, stopButton := gUI.DiG1.S7.bStop)
    Frame (926,191 285x149)
        shows ModuleDTD(enable := gUI.DiG1.bRVD1_enable, propPercent := gUI.DiG1.rRVD1Percent)
END_VISUALIZATION

// Device/Application/display/Module/ModuleX2
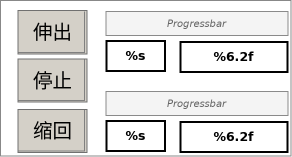
VISUALIZATION ModuleX2  // 292x157
VAR_IN_OUT
	extendButton		: BOOL;
	retractButton		: BOOL;
	stopButton			: BOOL;
	
	nameStr1			:STRING;
	posVal1				:REAL;
	percentBar1			:REAL;
	nameStr2			:STRING;
	posVal2				:REAL;
	percentBar2			:REAL;
END_VAR
    Group (5,5 285x150)
        Frame (0,0 85x150)
            shows OilBlock_PrimButton(extendButton := extendButton, retractButton := retractButton, stopButton := stopButton)
        Frame (95,0 190x70)
            shows OilBlock_PrimInfo(nameStr := nameStr1, posVal := posVal1, percentBar := percentBar1)
        Frame (95,80 190x70)
            shows OilBlock_PrimInfo(nameStr := nameStr2, posVal := posVal2, percentBar := percentBar2)
END_VISUALIZATION

// Device/Application/display/Module/ModuleX1
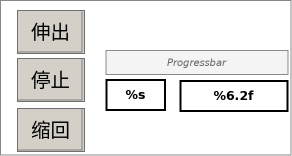
VISUALIZATION ModuleX1  // 292x156
VAR_IN_OUT
	extendButton		: BOOL;
	retractButton		: BOOL;
	stopButton			: BOOL;
	
	nameStr				:STRING;
	posVal				:REAL;
	percentBar			:REAL;
END_VAR
    Group (5,5 285x149)
        Frame (0,0 82x149)
            shows OilBlock_PrimButton(extendButton := extendButton, retractButton := retractButton, stopButton := stopButton)
        Frame (95,39 190x70)
            shows OilBlock_PrimInfo(nameStr := nameStr, posVal := posVal, percentBar := percentBar)
END_VISUALIZATION

// Device/Application/display/Module/ModuleX3
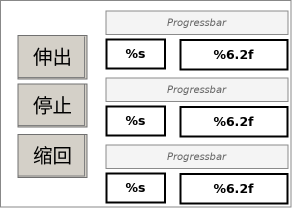
VISUALIZATION ModuleX3  // 292x208
VAR_IN_OUT
	extendButton		: BOOL;
	retractButton		: BOOL;
	stopButton			: BOOL;
	
	nameStr1			:STRING;
	posVal1				:REAL;
	percentBar1			:REAL;
	nameStr2			:STRING;
	posVal2				:REAL;
	percentBar2			:REAL;
	nameStr3			:STRING;
	posVal3				:REAL;
	percentBar3			:REAL;
END_VAR
    Group (5,5 285x201)
        Frame (0,25 85x150)
            shows OilBlock_PrimButton(extendButton := extendButton, retractButton := retractButton, stopButton := stopButton)
        Frame (95,0 190x67)
            shows OilBlock_PrimInfo(nameStr := nameStr1, posVal := posVal1, percentBar := percentBar1)
        Frame (95,67 190x67)
            shows OilBlock_PrimInfo(nameStr := nameStr2, posVal := posVal2, percentBar := percentBar2)
        Frame (95,134 190x67)
            shows OilBlock_PrimInfo(nameStr := nameStr3, posVal := posVal3, percentBar := percentBar3)
END_VISUALIZATION

// Device/Application/display/Module/ModuleX8
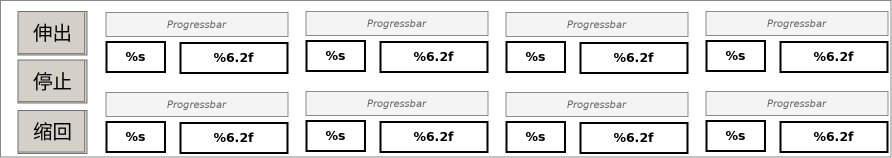
VISUALIZATION ModuleX8  // 892x158
VAR_IN_OUT
	extendButton		: BOOL;
	retractButton		: BOOL;
	stopButton			: BOOL;
	
	nameStr1			:STRING;
	posVal1				:REAL;
	percentBar1			:REAL;
	
	nameStr2			:STRING;
	posVal2				:REAL;
	percentBar2			:REAL;
	
	nameStr3			:STRING;
	posVal3				:REAL;
	percentBar3			:REAL;
	
	nameStr4			:STRING;
	posVal4				:REAL;
	percentBar4			:REAL;
	
	nameStr5			:STRING;
	posVal5				:REAL;
	percentBar5			:REAL;
	
	nameStr6			:STRING;
	posVal6				:REAL;
	percentBar6			:REAL;
	
	nameStr7			:STRING;
	posVal7				:REAL;
	percentBar7			:REAL;
	
	nameStr8			:STRING;
	posVal8				:REAL;
	percentBar8			:REAL;	
	
END_VAR
    Group (5,5 885x151)
        Frame (0,1 85x150)
            shows OilBlock_PrimButton(extendButton := extendButton, retractButton := retractButton, stopButton := stopButton)
        Group (95,0 390x151)
            Group (0,1 190x150)
                Frame (0,0 190x70)
                    shows OilBlock_PrimInfo(nameStr := nameStr1, posVal := posVal1, percentBar := percentBar1)
                Frame (0,80 190x70)
                    shows OilBlock_PrimInfo(nameStr := nameStr2, posVal := posVal2, percentBar := percentBar2)
            Frame (200,0 190x70)
                shows OilBlock_PrimInfo(nameStr := nameStr3, posVal := posVal3, percentBar := percentBar3)
            Frame (200,80 190x70)
                shows OilBlock_PrimInfo(nameStr := nameStr4, posVal := posVal4, percentBar := percentBar4)
        Frame (495,1 190x70)
            shows OilBlock_PrimInfo(nameStr := nameStr5, posVal := posVal5, percentBar := percentBar5)
        Frame (495,81 190x70)
            shows OilBlock_PrimInfo(nameStr := nameStr6, posVal := posVal6, percentBar := percentBar6)
        Frame (695,0 190x70)
            shows OilBlock_PrimInfo(nameStr := nameStr7, posVal := posVal7, percentBar := percentBar7)
        Frame (695,80 190x70)
            shows OilBlock_PrimInfo(nameStr := nameStr8, posVal := posVal8, percentBar := percentBar8)
END_VISUALIZATION

// Device/Application/display/Module/ModuleX4
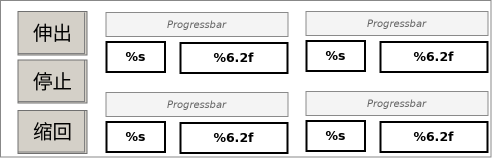
VISUALIZATION ModuleX4  // 492x158
VAR_IN_OUT
	extendButton		: BOOL;
	retractButton		: BOOL;
	stopButton			: BOOL;
	
	nameStr1			:STRING;
	posVal1				:REAL;
	percentBar1			:REAL;
	nameStr2			:STRING;
	posVal2				:REAL;
	percentBar2			:REAL;
	nameStr3			:STRING;
	posVal3				:REAL;
	percentBar3			:REAL;
	nameStr4			:STRING;
	posVal4				:REAL;
	percentBar4			:REAL;
	
	
END_VAR
    Group (5,5 485x151)
        Frame (0,1 85x150)
            shows OilBlock_PrimButton(extendButton := extendButton, retractButton := retractButton, stopButton := stopButton)
        Group (95,1 190x150)
            Frame (0,0 190x70)
                shows OilBlock_PrimInfo(nameStr := nameStr1, posVal := posVal1, percentBar := percentBar1)
            Frame (0,80 190x70)
                shows OilBlock_PrimInfo(nameStr := nameStr2, posVal := posVal2, percentBar := percentBar2)
        Frame (295,0 190x70)
            shows OilBlock_PrimInfo(nameStr := nameStr3, posVal := posVal3, percentBar := percentBar3)
        Frame (295,80 190x70)
            shows OilBlock_PrimInfo(nameStr := nameStr4, posVal := posVal4, percentBar := percentBar4)
END_VISUALIZATION

// Device/Application/display/Module/ModuleX5
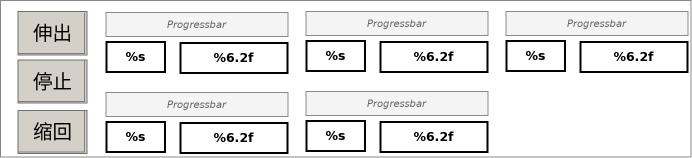
VISUALIZATION ModuleX5  // 692x158
VAR_IN_OUT
	extendButton		: BOOL;
	retractButton		: BOOL;
	stopButton			: BOOL;
	
	nameStr1			:STRING;
	posVal1				:REAL;
	percentBar1			:REAL;
	nameStr2			:STRING;
	posVal2				:REAL;
	percentBar2			:REAL;
	nameStr3			:STRING;
	posVal3				:REAL;
	percentBar3			:REAL;
	nameStr4			:STRING;
	posVal4				:REAL;
	percentBar4			:REAL;
	nameStr5			:STRING;
	posVal5				:REAL;
	percentBar5			:REAL;
	
	
END_VAR
    Group (5,5 685x151)
        Frame (0,1 85x150)
            shows OilBlock_PrimButton(extendButton := extendButton, retractButton := retractButton, stopButton := stopButton)
        Group (95,1 190x150)
            Frame (0,0 190x70)
                shows OilBlock_PrimInfo(nameStr := nameStr1, posVal := posVal1, percentBar := percentBar1)
            Frame (0,80 190x70)
                shows OilBlock_PrimInfo(nameStr := nameStr2, posVal := posVal2, percentBar := percentBar2)
        Frame (295,0 190x70)
            shows OilBlock_PrimInfo(nameStr := nameStr3, posVal := posVal3, percentBar := percentBar3)
        Frame (295,80 190x70)
            shows OilBlock_PrimInfo(nameStr := nameStr4, posVal := posVal4, percentBar := percentBar4)
        Frame (495,0 190x70)
            shows OilBlock_PrimInfo(nameStr := nameStr5, posVal := posVal5, percentBar := percentBar5)
END_VISUALIZATION

// Device/Application/display/OrigTi/Ceiling_Rail2
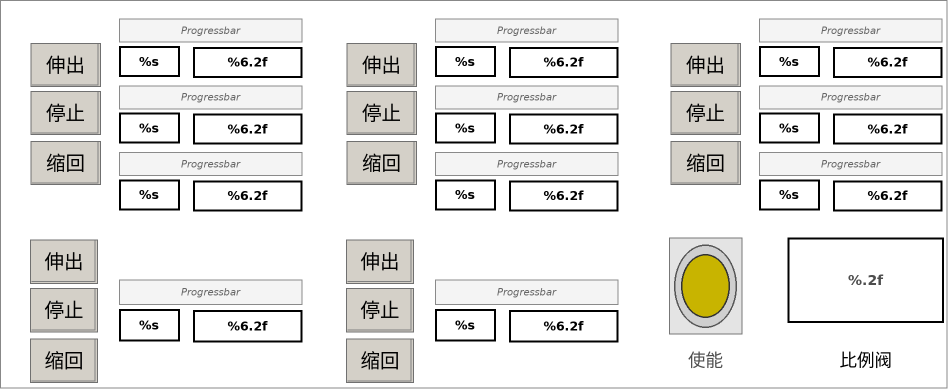
VISUALIZATION Ceiling_Rail2  // 948x389
    Frame (13,8 293x207)
        shows ModuleX3(extendButton := gUI.TiG.arrPV[2].sColumn[1].bExtend, retractButton := gUI.TiG.arrPV[2].sColumn[1].bRetract, stopButton := gUI.TiG.arrPV[2].sColumn[1].bStop, nameStr1 := gUI.TiG.arrPV[2].sNum[1].strName, posVal1 := gUI.TiG.arrPV[2].sNum[1].rPosition, percentBar1 := gUI.TiG.arrPV[2].sNum[1].rPercent, nameStr2 := gUI.TiG.arrPV[2].sNum[2].strName, posVal2 := gUI.TiG.arrPV[2].sNum[2].rPosition, percentBar2 := gUI.TiG.arrPV[2].sNum[2].rPercent, nameStr3 := gUI.TiG.arrPV[2].sNum[3].strName, posVal3 := gUI.TiG.arrPV[2].sNum[3].rPosition, percentBar3 := gUI.TiG.arrPV[2].sNum[3].rPercent)
    Frame (13,229 293x158)
        shows ModuleX1(extendButton := gUI.TiG.arrPV[2].sColumn[2].bExtend, retractButton := gUI.TiG.arrPV[2].sColumn[2].bRetract, stopButton := gUI.TiG.arrPV[2].sColumn[2].bStop, nameStr := gUI.TiG.arrPV[2].sNum[4].strName, posVal := gUI.TiG.arrPV[2].sNum[4].rPosition, percentBar := gUI.TiG.arrPV[2].sNum[4].rPercent)
    Frame (329,8 293x207)
        shows ModuleX3(extendButton := gUI.TiG.arrPV[2].sColumn[3].bExtend, retractButton := gUI.TiG.arrPV[2].sColumn[3].bRetract, stopButton := gUI.TiG.arrPV[2].sColumn[3].bStop, nameStr1 := gUI.TiG.arrPV[2].sNum[5].strName, posVal1 := gUI.TiG.arrPV[2].sNum[5].rPosition, percentBar1 := gUI.TiG.arrPV[2].sNum[5].rPercent, nameStr2 := gUI.TiG.arrPV[2].sNum[6].strName, posVal2 := gUI.TiG.arrPV[2].sNum[6].rPosition, percentBar2 := gUI.TiG.arrPV[2].sNum[6].rPercent, nameStr3 := gUI.TiG.arrPV[2].sNum[7].strName, posVal3 := gUI.TiG.arrPV[2].sNum[7].rPosition, percentBar3 := gUI.TiG.arrPV[2].sNum[7].rPercent)
    Frame (329,229 293x158)
        shows ModuleX1(extendButton := gUI.TiG.arrPV[2].sColumn[4].bExtend, retractButton := gUI.TiG.arrPV[2].sColumn[4].bRetract, stopButton := gUI.TiG.arrPV[2].sColumn[4].bStop, nameStr := gUI.TiG.arrPV[2].sNum[8].strName, posVal := gUI.TiG.arrPV[2].sNum[8].rPosition, percentBar := gUI.TiG.arrPV[2].sNum[8].rPercent)
    Frame (653,8 293x207)
        shows ModuleX3(extendButton := gUI.TiG.arrPV[2].sColumn[5].bExtend, retractButton := gUI.TiG.arrPV[2].sColumn[5].bRetract, stopButton := gUI.TiG.arrPV[2].sColumn[5].bStop, nameStr1 := gUI.TiG.arrPV[2].sNum[9].strName, posVal1 := gUI.TiG.arrPV[2].sNum[9].rPosition, percentBar1 := gUI.TiG.arrPV[2].sNum[9].rPercent, nameStr2 := gUI.TiG.arrPV[2].sNum[10].strName, posVal2 := gUI.TiG.arrPV[2].sNum[10].rPosition, percentBar2 := gUI.TiG.arrPV[2].sNum[10].rPercent, nameStr3 := gUI.TiG.arrPV[2].sNum[11].strName, posVal3 := gUI.TiG.arrPV[2].sNum[11].rPosition, percentBar3 := gUI.TiG.arrPV[2].sNum[11].rPercent)
    Frame (653,229 293x158)
        shows ModuleDTD(enable := gUI.TiG.arrPV[2].bPVD_enable, propPercent := gUI.TiG.arrPV[2].rPVDPercent)
END_VISUALIZATION

// Device/Application/display/Module/ModuleDTD
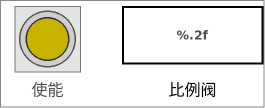
VISUALIZATION ModuleDTD  // 265x108
VAR_IN_OUT
	enable			:BOOL;
	propPercent		:REAL;
END_VAR
    Rectangle (122,6 141x58), "%.2f", text variable: propPercent
        OnMouseDown: write the text variable via Default, min 0, max 100
    Label (122,74 141x32), "比例阀"
    PushSwitchLed (13,6 69x66), variable: enable, behaviour: TOGGLE, style: Switch-PushSwitchLed-Yellow
    Label (13,74 69x32), "使能"
END_VISUALIZATION

// Device/Application/display/OrigDi/Floor_Rail_345
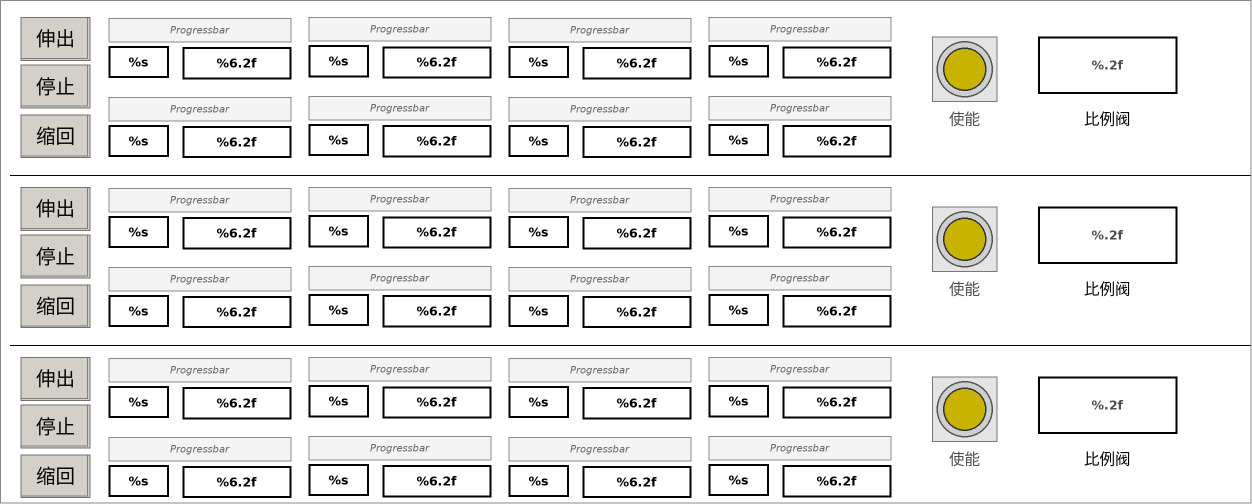
VISUALIZATION Floor_Rail_345  // 1252x504
    Frame (3,6 892x156)
        shows ModuleX8(extendButton := gUI.DiG.arrPV[3].sColumn[1].bExtend, retractButton := gUI.DiG.arrPV[3].sColumn[1].bRetract, stopButton := gUI.DiG.arrPV[3].sColumn[1].bStop, nameStr1 := gUI.DiG.arrPV[3].sNum[1].strName, posVal1 := gUI.DiG.arrPV[3].sNum[1].rPosition, percentBar1 := gUI.DiG.arrPV[3].sNum[1].rPercent, nameStr2 := gUI.DiG.arrPV[3].sNum[2].strName, posVal2 := gUI.DiG.arrPV[3].sNum[2].rPosition, percentBar2 := gUI.DiG.arrPV[3].sNum[2].rPercent, nameStr3 := gUI.DiG.arrPV[3].sNum[3].strName, posVal3 := gUI.DiG.arrPV[3].sNum[3].rPosition, percentBar3 := gUI.DiG.arrPV[3].sNum[3].rPercent, nameStr4 := gUI.DiG.arrPV[3].sNum[4].strName, posVal4 := gUI.DiG.arrPV[3].sNum[4].rPosition, percentBar4 := gUI.DiG.arrPV[3].sNum[4].rPercent, nameStr5 := gUI.DiG.arrPV[3].sNum[5].strName, posVal5 := gUI.DiG.arrPV[3].sNum[5].rPosition, percentBar5 := gUI.DiG.arrPV[3].sNum[5].rPercent, nameStr6 := gUI.DiG.arrPV[3].sNum[6].strName, posVal6 := gUI.DiG.arrPV[3].sNum[6].rPosition, percentBar6 := gUI.DiG.arrPV[3].sNum[6].rPercent, nameStr7 := gUI.DiG.arrPV[3].sNum[7].strName, posVal7 := gUI.DiG.arrPV[3].sNum[7].rPosition, percentBar7 := gUI.DiG.arrPV[3].sNum[7].rPercent, nameStr8 := gUI.DiG.arrPV[3].sNum[8].strName, posVal8 := gUI.DiG.arrPV[3].sNum[8].rPosition, percentBar8 := gUI.DiG.arrPV[3].sNum[8].rPercent)
    Frame (3,176 892x156)
        shows ModuleX8(extendButton := gUI.DiG.arrPV[4].sColumn[1].bExtend, retractButton := gUI.DiG.arrPV[4].sColumn[1].bRetract, stopButton := gUI.DiG.arrPV[4].sColumn[1].bStop, nameStr1 := gUI.DiG.arrPV[4].sNum[1].strName, posVal1 := gUI.DiG.arrPV[4].sNum[1].rPosition, percentBar1 := gUI.DiG.arrPV[4].sNum[1].rPercent, nameStr2 := gUI.DiG.arrPV[4].sNum[2].strName, posVal2 := gUI.DiG.arrPV[4].sNum[2].rPosition, percentBar2 := gUI.DiG.arrPV[4].sNum[2].rPercent, nameStr3 := gUI.DiG.arrPV[4].sNum[3].strName, posVal3 := gUI.DiG.arrPV[4].sNum[3].rPosition, percentBar3 := gUI.DiG.arrPV[4].sNum[3].rPercent, nameStr4 := gUI.DiG.arrPV[4].sNum[4].strName, posVal4 := gUI.DiG.arrPV[4].sNum[4].rPosition, percentBar4 := gUI.DiG.arrPV[4].sNum[4].rPercent, nameStr5 := gUI.DiG.arrPV[4].sNum[5].strName, posVal5 := gUI.DiG.arrPV[4].sNum[5].rPosition, percentBar5 := gUI.DiG.arrPV[4].sNum[5].rPercent, nameStr6 := gUI.DiG.arrPV[4].sNum[6].strName, posVal6 := gUI.DiG.arrPV[4].sNum[6].rPosition, percentBar6 := gUI.DiG.arrPV[4].sNum[6].rPercent, nameStr7 := gUI.DiG.arrPV[4].sNum[7].strName, posVal7 := gUI.DiG.arrPV[4].sNum[7].rPosition, percentBar7 := gUI.DiG.arrPV[4].sNum[7].rPercent, nameStr8 := gUI.DiG.arrPV[4].sNum[8].strName, posVal8 := gUI.DiG.arrPV[4].sNum[8].rPosition, percentBar8 := gUI.DiG.arrPV[4].sNum[8].rPercent)
    Frame (3,346 892x156)
        shows ModuleX8(extendButton := gUI.DiG.arrPV[5].sColumn[1].bExtend, retractButton := gUI.DiG.arrPV[5].sColumn[1].bStop, stopButton := gUI.DiG.arrPV[5].sColumn[1].bStop, nameStr1 := gUI.DiG.arrPV[5].sNum[1].strName, posVal1 := gUI.DiG.arrPV[5].sNum[1].rPosition, percentBar1 := gUI.DiG.arrPV[5].sNum[1].rPercent, nameStr2 := gUI.DiG.arrPV[5].sNum[2].strName, posVal2 := gUI.DiG.arrPV[5].sNum[2].rPosition, percentBar2 := gUI.DiG.arrPV[5].sNum[2].rPercent, nameStr3 := gUI.DiG.arrPV[5].sNum[3].strName, posVal3 := gUI.DiG.arrPV[5].sNum[3].rPosition, percentBar3 := gUI.DiG.arrPV[5].sNum[3].rPercent, nameStr4 := gUI.DiG.arrPV[5].sNum[4].strName, posVal4 := gUI.DiG.arrPV[5].sNum[4].rPosition, percentBar4 := gUI.DiG.arrPV[5].sNum[4].rPercent, nameStr5 := gUI.DiG.arrPV[5].sNum[5].strName, posVal5 := gUI.DiG.arrPV[5].sNum[5].rPosition, percentBar5 := gUI.DiG.arrPV[5].sNum[5].rPercent, nameStr6 := gUI.DiG.arrPV[5].sNum[6].strName, posVal6 := gUI.DiG.arrPV[5].sNum[6].rPosition, percentBar6 := gUI.DiG.arrPV[5].sNum[6].rPercent, nameStr7 := gUI.DiG.arrPV[5].sNum[7].strName, posVal7 := gUI.DiG.arrPV[5].sNum[7].rPosition, percentBar7 := gUI.DiG.arrPV[5].sNum[7].rPercent, nameStr8 := gUI.DiG.arrPV[5].sNum[8].strName, posVal8 := gUI.DiG.arrPV[5].sNum[8].rPosition, percentBar8 := gUI.DiG.arrPV[5].sNum[8].rPercent)
    Frame (918,31 261x106)
        shows ModuleDTD(enable := gUI.DiG.arrPV[3].bPVD_enable, propPercent := gUI.DiG.arrPV[3].rPVDPercent)
    Frame (918,201 261x106)
        shows ModuleDTD(enable := gUI.DiG.arrPV[4].bPVD_enable, propPercent := gUI.DiG.arrPV[4].rPVDPercent)
    Frame (918,371 261x106)
        shows ModuleDTD(enable := gUI.DiG.arrPV[5].bPVD_enable, propPercent := gUI.DiG.arrPV[5].rPVDPercent)
    Line (10,175) (1250,175)
    Line (10,345) (1250,345)
END_VISUALIZATION

// Device/Application/display/OrigDi/Floor_Rail6
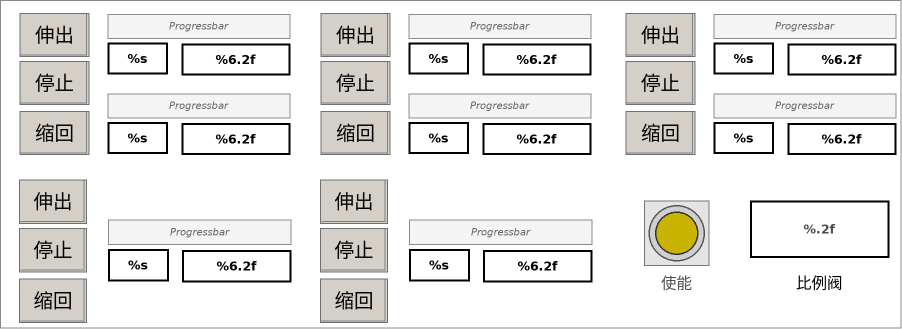
VISUALIZATION Floor_Rail6  // 902x329
    Frame (2,169 293x158)
        shows ModuleX1(extendButton := gUI.DiG.arrPV[6].sColumn[2].bExtend, retractButton := gUI.DiG.arrPV[6].sColumn[2].bRetract, stopButton := gUI.DiG.arrPV[6].sColumn[2].bStop, nameStr := gUI.DiG.arrPV[6].sNum[3].strName, posVal := gUI.DiG.arrPV[6].sNum[3].rPosition, percentBar := gUI.DiG.arrPV[6].sNum[3].rPercent)
    Frame (2,3 292x156)
        shows ModuleX2(extendButton := gUI.DiG.arrPV[6].sColumn[1].bExtend, retractButton := gUI.DiG.arrPV[6].sColumn[1].bRetract, stopButton := gUI.DiG.arrPV[6].sColumn[1].bStop, nameStr1 := gUI.DiG.arrPV[6].sNum[1].strName, posVal1 := gUI.DiG.arrPV[6].sNum[1].rPosition, percentBar1 := gUI.DiG.arrPV[6].sNum[1].rPercent, nameStr2 := gUI.DiG.arrPV[6].sNum[2].strName, posVal2 := gUI.DiG.arrPV[6].sNum[2].rPosition, percentBar2 := gUI.DiG.arrPV[6].sNum[2].rPercent)
    Frame (303,3 292x156)
        shows ModuleX2(extendButton := gUI.DiG.arrPV[6].sColumn[3].bExtend, retractButton := gUI.DiG.arrPV[6].sColumn[3].bRetract, stopButton := gUI.DiG.arrPV[6].sColumn[3].bStop, nameStr1 := gUI.DiG.arrPV[6].sNum[4].strName, posVal1 := gUI.DiG.arrPV[6].sNum[4].rPosition, percentBar1 := gUI.DiG.arrPV[6].sNum[4].rPercent, nameStr2 := gUI.DiG.arrPV[6].sNum[5].strName, posVal2 := gUI.DiG.arrPV[6].sNum[5].rPosition, percentBar2 := gUI.DiG.arrPV[6].sNum[5].rPercent)
    Frame (303,169 293x158)
        shows ModuleX1(extendButton := gUI.DiG.arrPV[6].sColumn[4].bExtend, retractButton := gUI.DiG.arrPV[6].sColumn[4].bRetract, stopButton := gUI.DiG.arrPV[6].sColumn[4].bStop, nameStr := gUI.DiG.arrPV[6].sNum[6].strName, posVal := gUI.DiG.arrPV[6].sNum[6].rPosition, percentBar := gUI.DiG.arrPV[6].sNum[6].rPercent)
    Frame (608,3 292x156)
        shows ModuleX2(extendButton := gUI.DiG.arrPV[6].sColumn[5].bExtend, retractButton := gUI.DiG.arrPV[6].sColumn[5].bRetract, stopButton := gUI.DiG.arrPV[6].sColumn[5].bStop, nameStr1 := gUI.DiG.arrPV[6].sNum[7].strName, posVal1 := gUI.DiG.arrPV[6].sNum[7].rPosition, percentBar1 := gUI.DiG.arrPV[6].sNum[7].rPercent, nameStr2 := gUI.DiG.arrPV[6].sNum[8].strName, posVal2 := gUI.DiG.arrPV[6].sNum[8].rPosition, percentBar2 := gUI.DiG.arrPV[6].sNum[8].rPercent)
    Frame (630,195 261x106)
        shows ModuleDTD(enable := gUI.DiG.arrPV[6].bPVD_enable, propPercent := gUI.DiG.arrPV[6].rPVDPercent)
END_VISUALIZATION

// Device/Application/display/OrigDi/Floor_Rail7
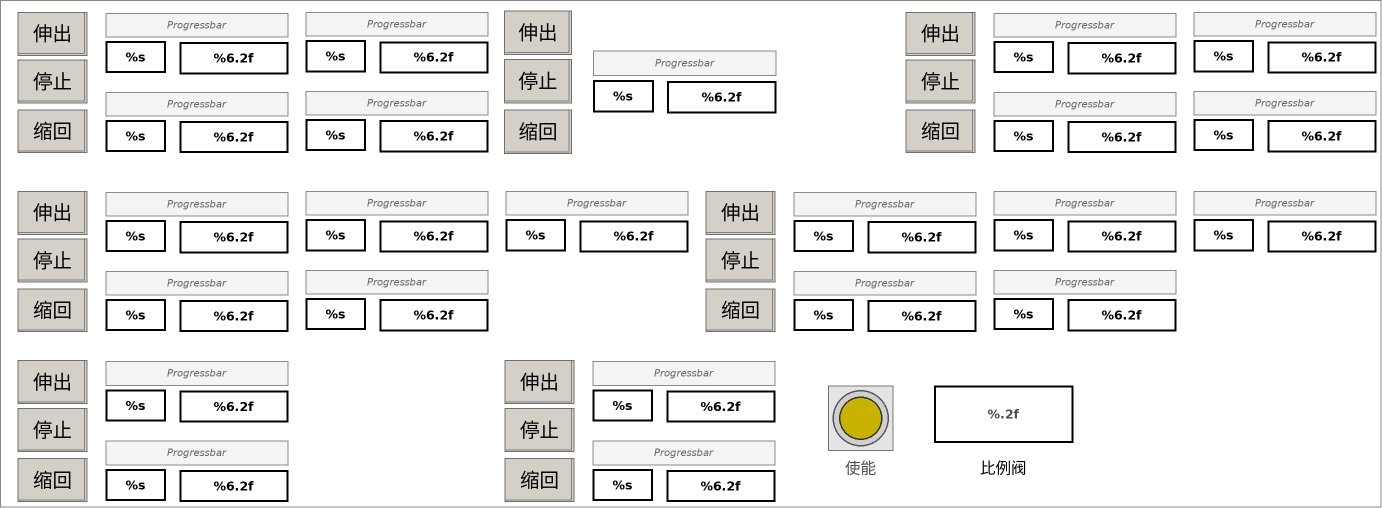
VISUALIZATION Floor_Rail7  // 1382x508
    Frame (0,1 492x156)
        shows ModuleX4(extendButton := gUI.DiG.arrPV[7].sColumn[1].bExtend, retractButton := gUI.DiG.arrPV[7].sColumn[1].bRetract, stopButton := gUI.DiG.arrPV[7].sColumn[1].bStop, nameStr1 := gUI.DiG.arrPV[7].sNum[1].strName, posVal1 := gUI.DiG.arrPV[7].sNum[1].rPosition, percentBar1 := gUI.DiG.arrPV[7].sNum[1].rPercent, nameStr2 := gUI.DiG.arrPV[7].sNum[2].strName, posVal2 := gUI.DiG.arrPV[7].sNum[2].rPosition, percentBar2 := gUI.DiG.arrPV[7].sNum[2].rPercent, nameStr3 := gUI.DiG.arrPV[7].sNum[3].strName, posVal3 := gUI.DiG.arrPV[7].sNum[3].rPosition, percentBar3 := gUI.DiG.arrPV[7].sNum[3].rPercent, nameStr4 := gUI.DiG.arrPV[7].sNum[4].strName, posVal4 := gUI.DiG.arrPV[7].sNum[4].rPosition, percentBar4 := gUI.DiG.arrPV[7].sNum[4].rPercent)
    Frame (487,0 293x158)
        shows ModuleX1(extendButton := gUI.DiG.arrPV[7].sColumn[2].bExtend, retractButton := gUI.DiG.arrPV[7].sColumn[2].bRetract, stopButton := gUI.DiG.arrPV[7].sColumn[2].bStop, nameStr := gUI.DiG.arrPV[7].sNum[5].strName, posVal := gUI.DiG.arrPV[7].sNum[5].rPosition, percentBar := gUI.DiG.arrPV[7].sNum[5].rPercent)
    Frame (888,1 492x156)
        shows ModuleX4(extendButton := gUI.DiG.arrPV[7].sColumn[3].bExtend, retractButton := gUI.DiG.arrPV[7].sColumn[3].bRetract, stopButton := gUI.DiG.arrPV[7].sColumn[3].bStop, nameStr1 := gUI.DiG.arrPV[7].sNum[6].strName, posVal1 := gUI.DiG.arrPV[7].sNum[6].rPosition, percentBar1 := gUI.DiG.arrPV[7].sNum[6].rPercent, nameStr2 := gUI.DiG.arrPV[7].sNum[7].strName, posVal2 := gUI.DiG.arrPV[7].sNum[7].rPosition, percentBar2 := gUI.DiG.arrPV[7].sNum[7].rPercent, nameStr3 := gUI.DiG.arrPV[7].sNum[8].strName, posVal3 := gUI.DiG.arrPV[7].sNum[8].rPosition, percentBar3 := gUI.DiG.arrPV[7].sNum[8].rPercent, nameStr4 := gUI.DiG.arrPV[7].sNum[9].strName, posVal4 := gUI.DiG.arrPV[7].sNum[9].rPosition, percentBar4 := gUI.DiG.arrPV[7].sNum[9].rPercent)
    Frame (0,180 692x156)
        shows ModuleX5(extendButton := gUI.DiG.arrPV[7].sColumn[4].bExtend, retractButton := gUI.DiG.arrPV[7].sColumn[4].bRetract, stopButton := gUI.DiG.arrPV[7].sColumn[4].bStop, nameStr1 := gUI.DiG.arrPV[7].sNum[10].strName, posVal1 := gUI.DiG.arrPV[7].sNum[10].rPosition, percentBar1 := gUI.DiG.arrPV[7].sNum[10].rPercent, nameStr2 := gUI.DiG.arrPV[7].sNum[11].strName, posVal2 := gUI.DiG.arrPV[7].sNum[11].rPosition, percentBar2 := gUI.DiG.arrPV[7].sNum[11].rPercent, nameStr3 := gUI.DiG.arrPV[7].sNum[12].strName, posVal3 := gUI.DiG.arrPV[7].sNum[12].rPosition, percentBar3 := gUI.DiG.arrPV[7].sNum[12].rPercent, nameStr4 := gUI.DiG.arrPV[7].sNum[13].strName, posVal4 := gUI.DiG.arrPV[7].sNum[13].rPosition, percentBar4 := gUI.DiG.arrPV[7].sNum[13].rPercent, nameStr5 := gUI.DiG.arrPV[7].sNum[14].strName, posVal5 := gUI.DiG.arrPV[7].sNum[14].rPosition, percentBar5 := gUI.DiG.arrPV[7].sNum[14].rPercent)
    Frame (688,180 692x156)
        shows ModuleX5(extendButton := gUI.DiG.arrPV[7].sColumn[5].bExtend, retractButton := gUI.DiG.arrPV[7].sColumn[5].bRetract, stopButton := gUI.DiG.arrPV[7].sColumn[5].bStop, nameStr1 := gUI.DiG.arrPV[7].sNum[15].strName, posVal1 := gUI.DiG.arrPV[7].sNum[15].rPosition, percentBar1 := gUI.DiG.arrPV[7].sNum[15].rPercent, nameStr2 := gUI.DiG.arrPV[7].sNum[16].strName, posVal2 := gUI.DiG.arrPV[7].sNum[16].rPosition, percentBar2 := gUI.DiG.arrPV[7].sNum[16].rPercent, nameStr3 := gUI.DiG.arrPV[7].sNum[17].strName, posVal3 := gUI.DiG.arrPV[7].sNum[17].rPosition, percentBar3 := gUI.DiG.arrPV[7].sNum[17].rPercent, nameStr4 := gUI.DiG.arrPV[7].sNum[18].strName, posVal4 := gUI.DiG.arrPV[7].sNum[18].rPosition, percentBar4 := gUI.DiG.arrPV[7].sNum[18].rPercent, nameStr5 := gUI.DiG.arrPV[7].sNum[19].strName, posVal5 := gUI.DiG.arrPV[7].sNum[19].rPosition, percentBar5 := gUI.DiG.arrPV[7].sNum[19].rPercent)
    Frame (0,350 292x156)
        shows ModuleX2(extendButton := gUI.DiG.arrPV[7].sColumn[6].bExtend, retractButton := gUI.DiG.arrPV[7].sColumn[6].bRetract, stopButton := gUI.DiG.arrPV[7].sColumn[6].bStop, nameStr1 := gUI.DiG.arrPV[7].sNum[20].strName, posVal1 := gUI.DiG.arrPV[7].sNum[20].rPosition, percentBar1 := gUI.DiG.arrPV[7].sNum[20].rPercent, nameStr2 := gUI.DiG.arrPV[7].sNum[21].strName, posVal2 := gUI.DiG.arrPV[7].sNum[21].rPosition, percentBar2 := gUI.DiG.arrPV[7].sNum[21].rPercent)
    Frame (487,350 292x156)
        shows ModuleX2(extendButton := gUI.DiG.arrPV[7].sColumn[7].bExtend, retractButton := gUI.DiG.arrPV[7].sColumn[7].bRetract, stopButton := gUI.DiG.arrPV[7].sColumn[7].bStop, nameStr1 := gUI.DiG.arrPV[7].sNum[22].strName, posVal1 := gUI.DiG.arrPV[7].sNum[22].rPosition, percentBar1 := gUI.DiG.arrPV[7].sNum[22].rPercent, nameStr2 := gUI.DiG.arrPV[7].sNum[23].strName, posVal2 := gUI.DiG.arrPV[7].sNum[23].rPosition, percentBar2 := gUI.DiG.arrPV[7].sNum[23].rPercent)
    Frame (814,380 261x106)
        shows ModuleDTD(enable := gUI.DiG.arrPV[7].bPVD_enable, propPercent := gUI.DiG.arrPV[7].rPVDPercent)
END_VISUALIZATION

// Device/Application/display/Module/old/Floor_Rail_12o
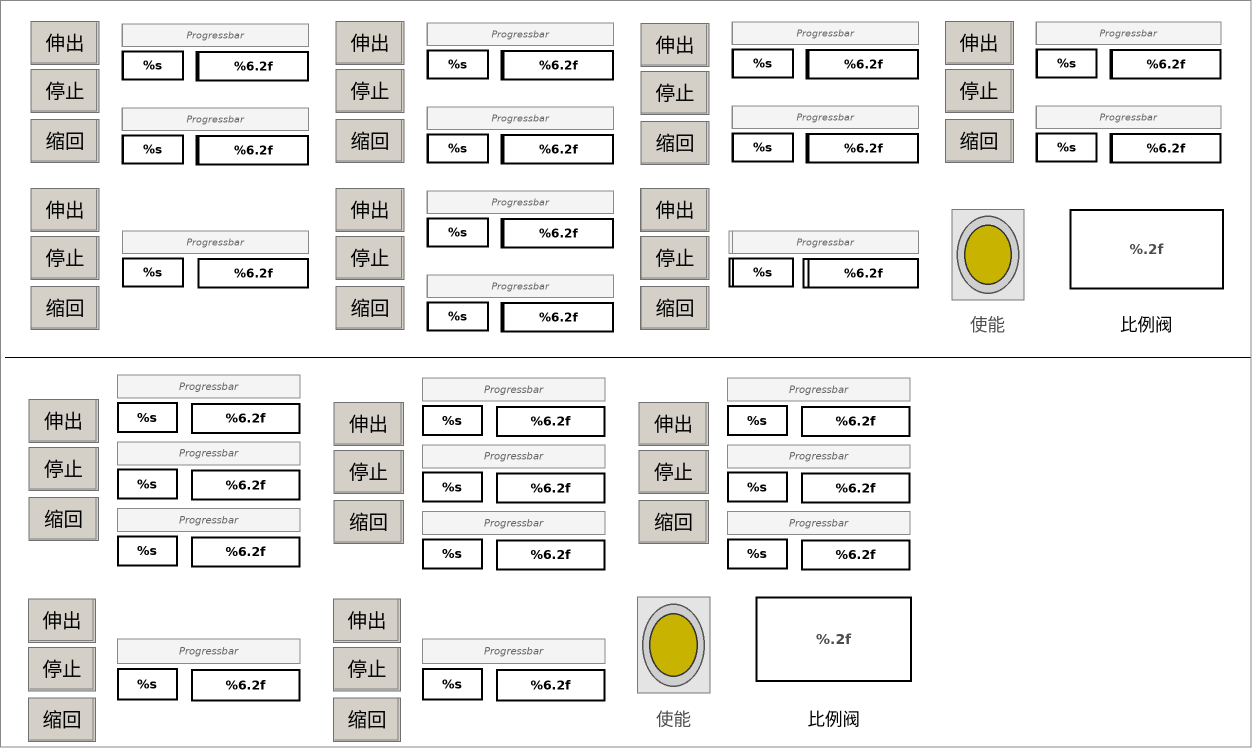
VISUALIZATION Floor_Rail_12o  // 1252x748
    Group (323,16 293x150)
        Group (98,1 195x149)
            Frame (0,0 190x65)
                shows OilBlock_PrimInfo(nameStr := gUI.DiG1.D28L1.strName, posVal := gUI.DiG1.D28L1.rPosition, percentBar := gUI.DiG1.D28L1.rPercent)
            Frame (0,84 190x65)
                shows OilBlock_PrimInfo(nameStr := gUI.DiG1.D28L2.strName, posVal := gUI.DiG1.D28L2.rPosition, percentBar := gUI.DiG1.D28L2.rPercent)
        Frame (0,0 84x149)
            shows OilBlock_PrimButton(extendButton := gUI.DiG1.S2.bExtend, retractButton := gUI.DiG1.S2.bRetract, stopButton := gUI.DiG1.S2.bStop)
    Group (421,17 195x149)
        Frame (0,0 195x65)
            shows OilBlock_PrimInfo(nameStr := gUI.DiG1.D28L1.strName, posVal := gUI.DiG1.D28L1.rPosition, percentBar := gUI.DiG1.D28L1.rPercent)
        Frame (0,84 195x65)
            shows OilBlock_PrimInfo(nameStr := gUI.DiG1.D28L2.strName, posVal := gUI.DiG1.D28L2.rPosition, percentBar := gUI.DiG1.D28L2.rPercent)
    Frame (421,17 195x65)
        shows OilBlock_PrimInfo(nameStr := gUI.DiG1.D28L1.strName, posVal := gUI.DiG1.D28L1.rPosition, percentBar := gUI.DiG1.D28L1.rPercent)
    Frame (421,101 195x65)
        shows OilBlock_PrimInfo(nameStr := gUI.DiG1.D28L2.strName, posVal := gUI.DiG1.D28L2.rPosition, percentBar := gUI.DiG1.D28L2.rPercent)
    Frame (323,16 84x149)
        shows OilBlock_PrimButton(extendButton := gUI.DiG1.S2.bExtend, retractButton := gUI.DiG1.S2.bRetract, stopButton := gUI.DiG1.S2.bStop)
    Group (18,16 293x151)
        Frame (0,0 84x149)
            shows OilBlock_PrimButton(extendButton := gUI.DiG1.S1.bExtend, retractButton := gUI.DiG1.S1.bRetract, stopButton := gUI.DiG1.S1.bStop)
        Group (98,2 195x149)
            Frame (0,0 190x65)
                shows OilBlock_PrimInfo(nameStr := gUI.DiG1.D00Q1.strName, posVal := gUI.DiG1.D00Q1.rPosition, percentBar := gUI.DiG1.D00Q1.rPercent)
            Frame (0,84 190x65)
                shows OilBlock_PrimInfo(nameStr := gUI.DiG1.D00Q2.strName, posVal := gUI.DiG1.D00Q2.rPosition, percentBar := gUI.DiG1.D00Q2.rPercent)
    Frame (18,16 84x149)
        shows OilBlock_PrimButton(extendButton := gUI.DiG1.S1.bExtend, retractButton := gUI.DiG1.S1.bRetract, stopButton := gUI.DiG1.S1.bStop)
    Group (116,18 195x149)
        Frame (0,0 195x65)
            shows OilBlock_PrimInfo(nameStr := gUI.DiG1.D00Q1.strName, posVal := gUI.DiG1.D00Q1.rPosition, percentBar := gUI.DiG1.D00Q1.rPercent)
        Frame (0,84 195x65)
            shows OilBlock_PrimInfo(nameStr := gUI.DiG1.D00Q2.strName, posVal := gUI.DiG1.D00Q2.rPosition, percentBar := gUI.DiG1.D00Q2.rPercent)
    Frame (116,18 195x65)
        shows OilBlock_PrimInfo(nameStr := gUI.DiG1.D00Q1.strName, posVal := gUI.DiG1.D00Q1.rPosition, percentBar := gUI.DiG1.D00Q1.rPercent)
    Frame (116,102 195x65)
        shows OilBlock_PrimInfo(nameStr := gUI.DiG1.D00Q2.strName, posVal := gUI.DiG1.D00Q2.rPosition, percentBar := gUI.DiG1.D00Q2.rPercent)
    Group (18,183 293x149)
        Frame (98,42 195x65)
            shows OilBlock_PrimInfo(nameStr := gUI.DiG1.D01L.strName, posVal := gUI.DiG1.D01L.rPosition, percentBar := gUI.DiG1.D01L.rPercent)
        Frame (0,0 84x149)
            shows OilBlock_PrimButton(extendButton := gUI.DiG1.S5.bExtend, retractButton := gUI.DiG1.S5.bRetract, stopButton := gUI.DiG1.S5.bStop)
    Frame (116,225 195x65)
        shows OilBlock_PrimInfo(nameStr := gUI.DiG1.D01L.strName, posVal := gUI.DiG1.D01L.rPosition, percentBar := gUI.DiG1.D01L.rPercent)
    Frame (18,183 84x149)
        shows OilBlock_PrimButton(extendButton := gUI.DiG1.S5.bExtend, retractButton := gUI.DiG1.S5.bRetract, stopButton := gUI.DiG1.S5.bStop)
    Group (323,183 293x151)
        Group (98,2 195x149)
            Frame (0,0 190x65)
                shows OilBlock_PrimInfo(nameStr := gUI.DiG1.D28Q.strName, posVal := gUI.DiG1.D28Q.rPosition, percentBar := gUI.DiG1.D28Q.rPercent)
            Frame (0,84 190x65)
                shows OilBlock_PrimInfo(nameStr := gUI.DiG1.D29Q.strName, posVal := gUI.DiG1.D29Q.rPosition, percentBar := gUI.DiG1.D29Q.rPercent)
        Frame (0,0 84x149)
            shows OilBlock_PrimButton(extendButton := gUI.DiG1.S6.bExtend, retractButton := gUI.DiG1.S6.bRetract, stopButton := gUI.DiG1.S6.bStop)
    Group (421,185 195x149)
        Frame (0,0 195x65)
            shows OilBlock_PrimInfo(nameStr := gUI.DiG1.D28Q.strName, posVal := gUI.DiG1.D28Q.rPosition, percentBar := gUI.DiG1.D28Q.rPercent)
        Frame (0,84 195x65)
            shows OilBlock_PrimInfo(nameStr := gUI.DiG1.D29Q.strName, posVal := gUI.DiG1.D29Q.rPosition, percentBar := gUI.DiG1.D29Q.rPercent)
    Frame (421,185 195x65)
        shows OilBlock_PrimInfo(nameStr := gUI.DiG1.D28Q.strName, posVal := gUI.DiG1.D28Q.rPosition, percentBar := gUI.DiG1.D28Q.rPercent)
    Frame (421,269 195x65)
        shows OilBlock_PrimInfo(nameStr := gUI.DiG1.D29Q.strName, posVal := gUI.DiG1.D29Q.rPosition, percentBar := gUI.DiG1.D29Q.rPercent)
    Frame (323,183 84x149)
        shows OilBlock_PrimButton(extendButton := gUI.DiG1.S6.bExtend, retractButton := gUI.DiG1.S6.bRetract, stopButton := gUI.DiG1.S6.bStop)
    Group (628,16 293x151)
        Group (98,0 195x149)
            Frame (0,0 190x65)
                shows OilBlock_PrimInfo(nameStr := gUI.DiG1.D29L.strName, posVal := gUI.DiG1.D29L.rPosition, percentBar := gUI.DiG1.D29L.rPercent)
            Frame (0,84 190x65)
                shows OilBlock_PrimInfo(nameStr := gUI.DiG1.D30L.strName, posVal := gUI.DiG1.D30L.rPosition, percentBar := gUI.DiG1.D30L.rPercent)
        Frame (0,2 84x149)
            shows OilBlock_PrimButton(extendButton := gUI.DiG1.S3.bExtend, retractButton := gUI.DiG1.S3.bRetract, stopButton := gUI.DiG1.S3.bStop)
    Group (726,16 195x149)
        Frame (0,0 195x65)
            shows OilBlock_PrimInfo(nameStr := gUI.DiG1.D29L.strName, posVal := gUI.DiG1.D29L.rPosition, percentBar := gUI.DiG1.D29L.rPercent)
        Frame (0,84 195x65)
            shows OilBlock_PrimInfo(nameStr := gUI.DiG1.D30L.strName, posVal := gUI.DiG1.D30L.rPosition, percentBar := gUI.DiG1.D30L.rPercent)
    Frame (726,16 195x65)
        shows OilBlock_PrimInfo(nameStr := gUI.DiG1.D29L.strName, posVal := gUI.DiG1.D29L.rPosition, percentBar := gUI.DiG1.D29L.rPercent)
    Frame (726,100 195x65)
        shows OilBlock_PrimInfo(nameStr := gUI.DiG1.D30L.strName, posVal := gUI.DiG1.D30L.rPosition, percentBar := gUI.DiG1.D30L.rPercent)
    Frame (628,18 84x149)
        shows OilBlock_PrimButton(extendButton := gUI.DiG1.S3.bExtend, retractButton := gUI.DiG1.S3.bRetract, stopButton := gUI.DiG1.S3.bStop)
    Group (628,183 293x149)
        Group (0,0 293x149)
            Frame (95,42 190x65)
                shows OilBlock_PrimInfo(nameStr := gUI.DiG1.D30Q.strName, posVal := gUI.DiG1.D30Q.rPosition, percentBar := gUI.DiG1.D30Q.rPercent)
            Frame (0,0 82x149)
                shows OilBlock_PrimButton(extendButton := gUI.DiG1.S7.bExtend, retractButton := gUI.DiG1.S7.bRetract, stopButton := gUI.DiG1.S7.bStop)
        Frame (98,42 195x65)
            shows OilBlock_PrimInfo(nameStr := gUI.DiG1.D30Q.strName, posVal := gUI.DiG1.D30Q.rPosition, percentBar := gUI.DiG1.D30Q.rPercent)
        Frame (0,0 84x149)
            shows OilBlock_PrimButton(extendButton := gUI.DiG1.S7.bExtend, retractButton := gUI.DiG1.S7.bRetract, stopButton := gUI.DiG1.S7.bStop)
    Group (933,16 290x149)
        Group (97,0 193x149)
            Frame (0,0 190x65)
                shows OilBlock_PrimInfo(nameStr := gUI.DiG1.D00L1.strName, posVal := gUI.DiG1.D00L1.rPosition, percentBar := gUI.DiG1.D00L1.rPercent)
            Frame (0,84 190x65)
                shows OilBlock_PrimInfo(nameStr := gUI.DiG1.D00L2.strName, posVal := gUI.DiG1.D00L2.rPosition, percentBar := gUI.DiG1.D00L2.rPercent)
        Frame (0,0 83x149)
            shows OilBlock_PrimButton(extendButton := gUI.DiG1.S4.bExtend, retractButton := gUI.DiG1.S4.bRetract, stopButton := gUI.DiG1.S4.bStop)
    Group (1030,16 193x149)
        Frame (0,0 193x65)
            shows OilBlock_PrimInfo(nameStr := gUI.DiG1.D00L1.strName, posVal := gUI.DiG1.D00L1.rPosition, percentBar := gUI.DiG1.D00L1.rPercent)
        Frame (0,84 193x65)
            shows OilBlock_PrimInfo(nameStr := gUI.DiG1.D00L2.strName, posVal := gUI.DiG1.D00L2.rPosition, percentBar := gUI.DiG1.D00L2.rPercent)
    Frame (1030,16 193x65)
        shows OilBlock_PrimInfo(nameStr := gUI.DiG1.D00L1.strName, posVal := gUI.DiG1.D00L1.rPosition, percentBar := gUI.DiG1.D00L1.rPercent)
    Frame (1030,100 193x65)
        shows OilBlock_PrimInfo(nameStr := gUI.DiG1.D00L2.strName, posVal := gUI.DiG1.D00L2.rPosition, percentBar := gUI.DiG1.D00L2.rPercent)
    Frame (933,16 83x149)
        shows OilBlock_PrimButton(extendButton := gUI.DiG1.S4.bExtend, retractButton := gUI.DiG1.S4.bRetract, stopButton := gUI.DiG1.S4.bStop)
    Frame (936,201 290x149)
        shows ModuleDTD(enable := gUI.DiG1.bRVD1_enable, propPercent := gUI.DiG1.rRVD1Percent)
    Frame (11,364 293x207)
        shows ModuleX3(extendButton := gUI.DiG2.S1.bExtend, retractButton := gUI.DiG2.S1.bRetract, stopButton := gUI.DiG2.S1.bStop, nameStr1 := gUI.DiG2.D02L.strName, posVal1 := gUI.DiG2.D02L.rPosition, percentBar1 := gUI.DiG2.D02L.rPercent, nameStr2 := gUI.DiG2.D03L.strName, posVal2 := gUI.DiG2.D03L.rPosition, percentBar2 := gUI.DiG2.D03L.rPercent, nameStr3 := gUI.DiG2.D04L.strName, posVal3 := gUI.DiG2.D04L.rPosition, percentBar3 := gUI.DiG2.D04L.rPercent)
    Frame (11,588 293x158)
        shows ModuleX1(extendButton := gUI.DiG2.S2.bExtend, retractButton := gUI.DiG2.S2.bRetract, stopButton := gUI.DiG2.S2.bStop, nameStr := gUI.DiG2.D05L.strName, posVal := gUI.DiG2.D05L.rPosition, percentBar := gUI.DiG2.D05L.rPercent)
    Frame (316,367 293x207)
        shows ModuleX3(extendButton := gUI.DiG2.S3.bExtend, retractButton := gUI.DiG2.S3.bRetract, stopButton := gUI.DiG2.S3.bStop, nameStr1 := gUI.DiG2.D06L.strName, posVal1 := gUI.DiG2.D06L.rPosition, percentBar1 := gUI.DiG2.D06L.rPercent, nameStr2 := gUI.DiG2.D07L.strName, posVal2 := gUI.DiG2.D07L.rPosition, percentBar2 := gUI.DiG2.D07L.rPercent, nameStr3 := gUI.DiG2.D08L.strName, posVal3 := gUI.DiG2.D08L.rPosition, percentBar3 := gUI.DiG2.D08L.rPercent)
    Frame (316,588 293x158)
        shows ModuleX1(extendButton := gUI.DiG2.S4.bExtend, retractButton := gUI.DiG2.S4.bRetract, stopButton := gUI.DiG2.S4.bStop, nameStr := gUI.DiG2.D09L.strName, posVal := gUI.DiG2.D09L.rPosition, percentBar := gUI.DiG2.D09L.rPercent)
    Frame (621,367 293x207)
        shows ModuleX3(extendButton := gUI.DiG2.S5.bExtend, retractButton := gUI.DiG2.S5.bRetract, stopButton := gUI.DiG2.S5.bStop, nameStr1 := gUI.DiG2.D10L.strName, posVal1 := gUI.DiG2.D10L.rPosition, percentBar1 := gUI.DiG2.D10L.rPercent, nameStr2 := gUI.DiG2.D11L.strName, posVal2 := gUI.DiG2.D11L.rPosition, percentBar2 := gUI.DiG2.D11L.rPercent, nameStr3 := gUI.DiG2.D12L.strName, posVal3 := gUI.DiG2.D12L.rPosition, percentBar3 := gUI.DiG2.D12L.rPercent)
    Frame (621,588 293x158)
        shows ModuleDTD(enable := gUI.DiG2.bRVD2_enable, propPercent := gUI.DiG2.rRVD2Percent)
    Line (5,357) (1250,357)
END_VISUALIZATION

// Device/Application/display/OrigDi/Floor_Rail1
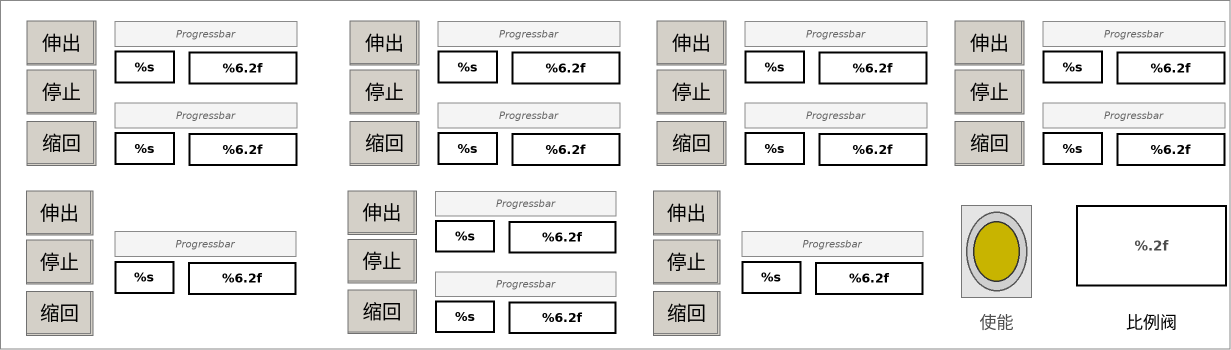
VISUALIZATION Floor_Rail1  // 1231x350
    Frame (9,10 292x160)
        shows ModuleX2(extendButton := gUI.DiG.arrPV[1].sColumn[1].bExtend, retractButton := gUI.DiG.arrPV[1].sColumn[1].bRetract, stopButton := gUI.DiG.arrPV[1].sColumn[1].bStop, nameStr1 := gUI.DiG.arrPV[1].sNum[1].strName, posVal1 := gUI.DiG.arrPV[1].sNum[1].rPosition, percentBar1 := gUI.DiG.arrPV[1].sNum[1].rPercent, nameStr2 := gUI.DiG.arrPV[1].sNum[2].strName, posVal2 := gUI.DiG.arrPV[1].sNum[2].rPosition, percentBar2 := gUI.DiG.arrPV[1].sNum[2].rPercent)
    Frame (332,10 292x160)
        shows ModuleX2(extendButton := gUI.DiG.arrPV[1].sColumn[2].bExtend, retractButton := gUI.DiG.arrPV[1].sColumn[2].bRetract, stopButton := gUI.DiG.arrPV[1].sColumn[2].bStop, nameStr1 := gUI.DiG.arrPV[1].sNum[3].strName, posVal1 := gUI.DiG.arrPV[1].sNum[3].rPosition, percentBar1 := gUI.DiG.arrPV[1].sNum[3].rPercent, nameStr2 := gUI.DiG.arrPV[1].sNum[4].strName, posVal2 := gUI.DiG.arrPV[1].sNum[4].rPosition, percentBar2 := gUI.DiG.arrPV[1].sNum[4].rPercent)
    Frame (639,10 292x160)
        shows ModuleX2(extendButton := gUI.DiG.arrPV[1].sColumn[3].bExtend, retractButton := gUI.DiG.arrPV[1].sColumn[3].bRetract, stopButton := gUI.DiG.arrPV[1].sColumn[3].bStop, nameStr1 := gUI.DiG.arrPV[1].sNum[5].strName, posVal1 := gUI.DiG.arrPV[1].sNum[5].rPosition, percentBar1 := gUI.DiG.arrPV[1].sNum[5].rPercent, nameStr2 := gUI.DiG.arrPV[1].sNum[6].strName, posVal2 := gUI.DiG.arrPV[1].sNum[6].rPosition, percentBar2 := gUI.DiG.arrPV[1].sNum[6].rPercent)
    Frame (937,10 292x160)
        shows ModuleX2(extendButton := gUI.DiG.arrPV[1].sColumn[4].bExtend, retractButton := gUI.DiG.arrPV[1].sColumn[4].bRetract, stopButton := gUI.DiG.arrPV[1].sColumn[4].bStop, nameStr1 := gUI.DiG.arrPV[1].sNum[7].strName, posVal1 := gUI.DiG.arrPV[1].sNum[7].rPosition, percentBar1 := gUI.DiG.arrPV[1].sNum[7].rPercent, nameStr2 := gUI.DiG.arrPV[1].sNum[8].strName, posVal2 := gUI.DiG.arrPV[1].sNum[8].rPosition, percentBar2 := gUI.DiG.arrPV[1].sNum[8].rPercent)
    Frame (946,197 283x151)
        shows ModuleDTD(enable := gUI.DiG.arrPV[1].bPVD_enable, propPercent := gUI.DiG.arrPV[1].rPVDPercent)
    Frame (9,180 291x160)
        shows ModuleX1(extendButton := gUI.DiG.arrPV[1].sColumn[5].bExtend, retractButton := gUI.DiG.arrPV[1].sColumn[5].bRetract, stopButton := gUI.DiG.arrPV[1].sColumn[5].bStop, nameStr := gUI.DiG.arrPV[1].sNum[9].strName, posVal := gUI.DiG.arrPV[1].sNum[9].rPosition, percentBar := gUI.DiG.arrPV[1].sNum[9].rPercent)
    Frame (636,180 291x160)
        shows ModuleX1(extendButton := gUI.DiG.arrPV[1].sColumn[7].bExtend, retractButton := gUI.DiG.arrPV[1].sColumn[7].bRetract, stopButton := gUI.DiG.arrPV[1].sColumn[7].bStop, nameStr := gUI.DiG.arrPV[1].sNum[12].strName, posVal := gUI.DiG.arrPV[1].sNum[12].rPosition, percentBar := gUI.DiG.arrPV[1].sNum[12].rPercent)
    Frame (330,180 290x158)
        shows ModuleX2(extendButton := gUI.DiG.arrPV[1].sColumn[6].bExtend, retractButton := gUI.DiG.arrPV[1].sColumn[6].bRetract, stopButton := gUI.DiG.arrPV[1].sColumn[6].bStop, nameStr1 := gUI.DiG.arrPV[1].sNum[10].strName, posVal1 := gUI.DiG.arrPV[1].sNum[10].rPosition, percentBar1 := gUI.DiG.arrPV[1].sNum[10].rPercent, nameStr2 := gUI.DiG.arrPV[1].sNum[11].strName, posVal2 := gUI.DiG.arrPV[1].sNum[11].rPosition, percentBar2 := gUI.DiG.arrPV[1].sNum[11].rPercent)
END_VISUALIZATION

// Device/Application/display/OrigDi/Floor_Rail_12
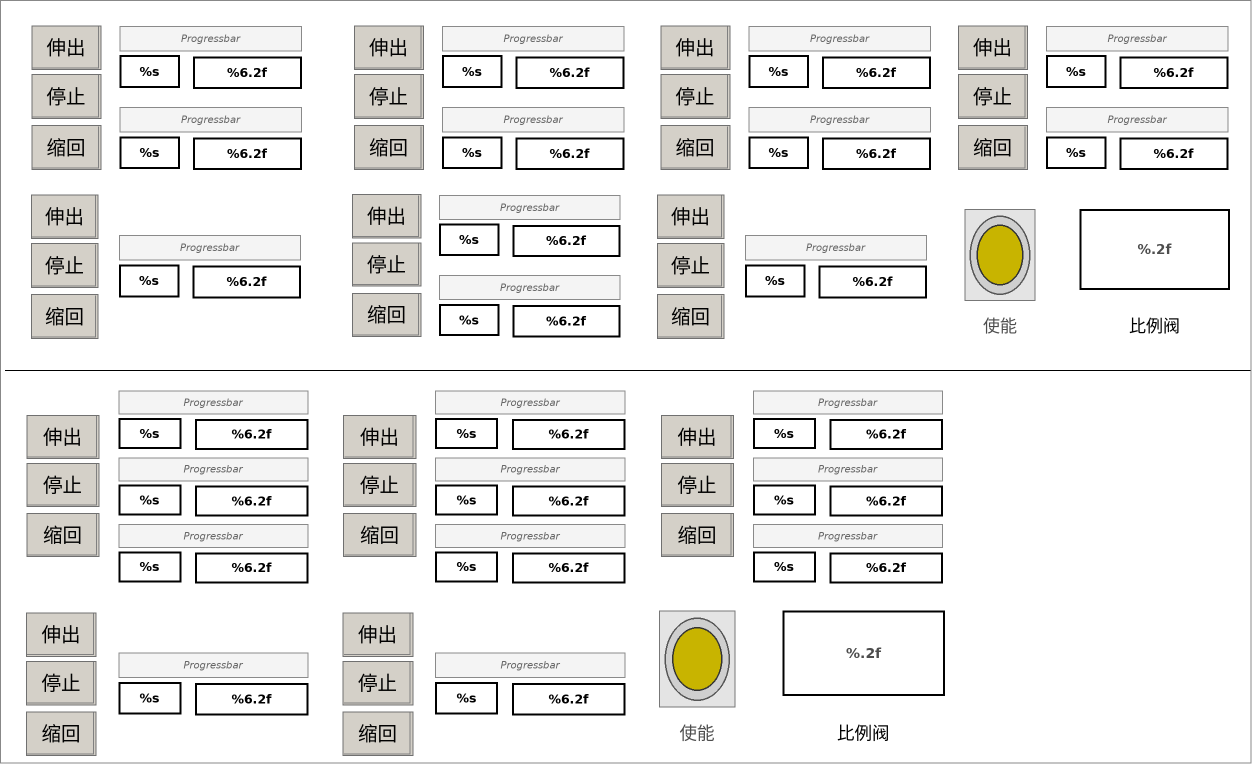
VISUALIZATION Floor_Rail_12  // 1252x764
    Frame (5,5 1229x348)
        shows Floor_Rail1()
    Frame (3,375 946x387)
        shows Floor_Rail2()
    Line (5,370) (1250,370)
END_VISUALIZATION

// Device/Application/display/OrigDi/Floor_Rail_67
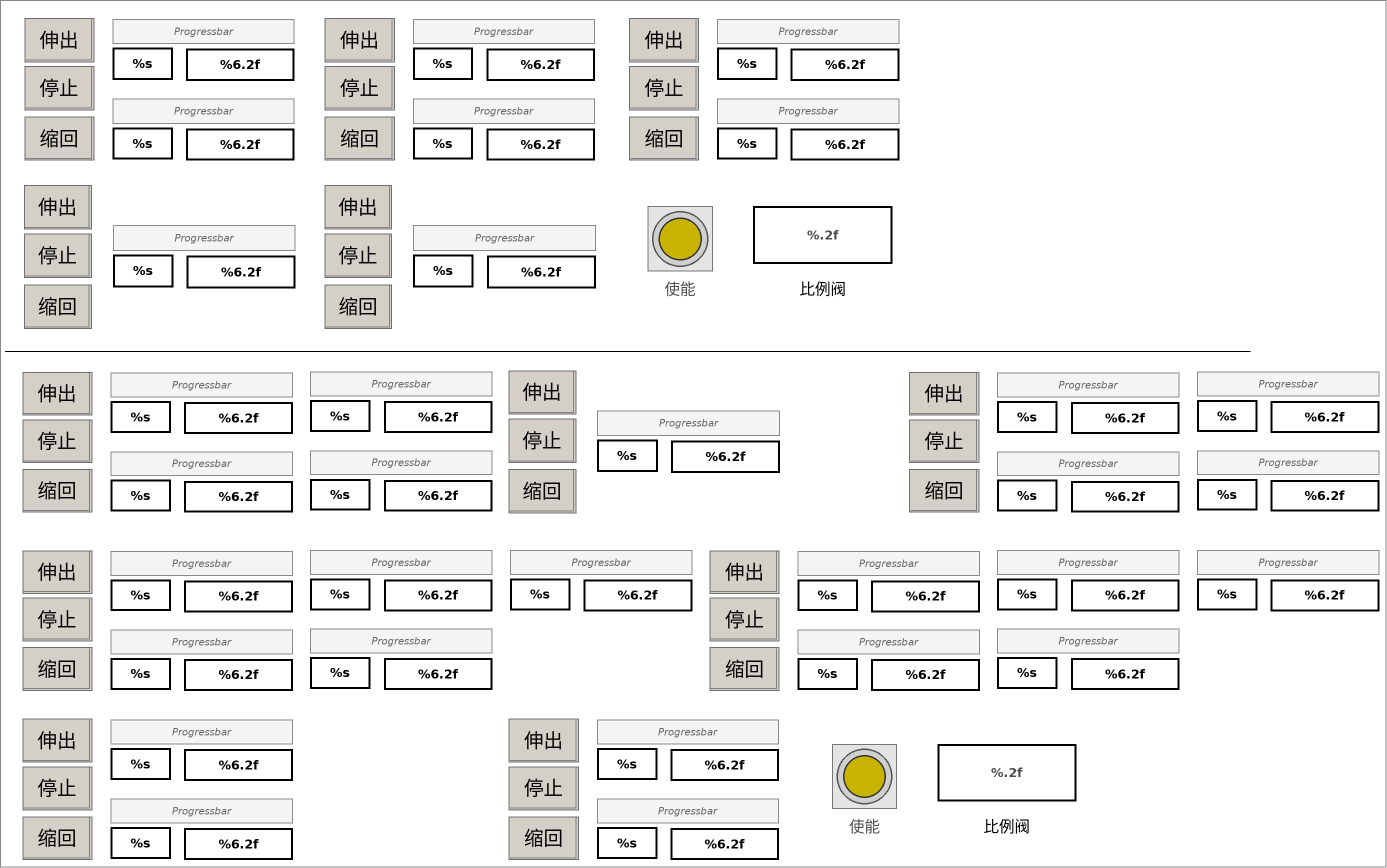
VISUALIZATION Floor_Rail_67  // 1387x868
    Frame (5,5 900x330)
        shows Floor_Rail6()
    Frame (5,360 1380x506)
        shows Floor_Rail7()
    Line (5,351) (1250,351)
END_VISUALIZATION

// Device/Application/display/OrigDi/Floor_Rail7_ByNum
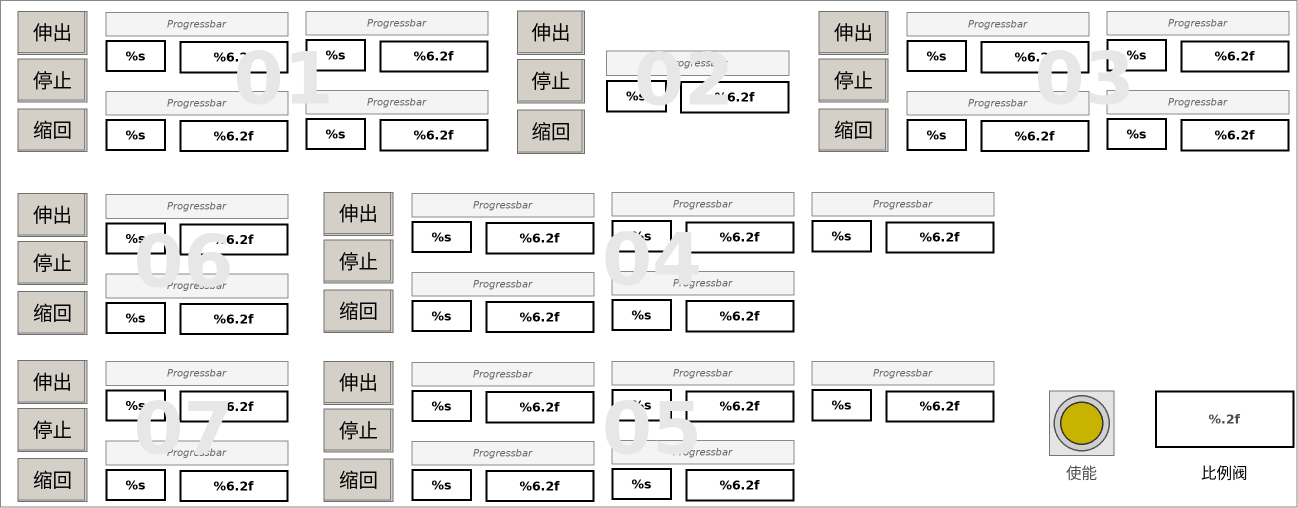
VISUALIZATION Floor_Rail7_ByNum  // 1298x508
    Frame (0,0 492x156), "01"
        shows ModuleX4(extendButton := gUI.DiG.arrPV[7].sColumn[1].bExtend, retractButton := gUI.DiG.arrPV[7].sColumn[1].bRetract, stopButton := gUI.DiG.arrPV[7].sColumn[1].bStop, nameStr1 := gUI.DiG.arrPV[7].sNum[1].strName, posVal1 := gUI.DiG.arrPV[7].sNum[1].rPosition, percentBar1 := gUI.DiG.arrPV[7].sNum[1].rPercent, nameStr2 := gUI.DiG.arrPV[7].sNum[2].strName, posVal2 := gUI.DiG.arrPV[7].sNum[2].rPosition, percentBar2 := gUI.DiG.arrPV[7].sNum[2].rPercent, nameStr3 := gUI.DiG.arrPV[7].sNum[3].strName, posVal3 := gUI.DiG.arrPV[7].sNum[3].rPosition, percentBar3 := gUI.DiG.arrPV[7].sNum[3].rPercent, nameStr4 := gUI.DiG.arrPV[7].sNum[4].strName, posVal4 := gUI.DiG.arrPV[7].sNum[4].rPosition, percentBar4 := gUI.DiG.arrPV[7].sNum[4].rPercent)
    Frame (500,0 293x158), "02"
        shows ModuleX1(extendButton := gUI.DiG.arrPV[7].sColumn[2].bExtend, retractButton := gUI.DiG.arrPV[7].sColumn[2].bRetract, stopButton := gUI.DiG.arrPV[7].sColumn[2].bStop, nameStr := gUI.DiG.arrPV[7].sNum[5].strName, posVal := gUI.DiG.arrPV[7].sNum[5].rPosition, percentBar := gUI.DiG.arrPV[7].sNum[5].rPercent)
    Frame (801,0 492x156), "03"
        shows ModuleX4(extendButton := gUI.DiG.arrPV[7].sColumn[3].bExtend, retractButton := gUI.DiG.arrPV[7].sColumn[3].bRetract, stopButton := gUI.DiG.arrPV[7].sColumn[3].bStop, nameStr1 := gUI.DiG.arrPV[7].sNum[6].strName, posVal1 := gUI.DiG.arrPV[7].sNum[6].rPosition, percentBar1 := gUI.DiG.arrPV[7].sNum[6].rPercent, nameStr2 := gUI.DiG.arrPV[7].sNum[7].strName, posVal2 := gUI.DiG.arrPV[7].sNum[7].rPosition, percentBar2 := gUI.DiG.arrPV[7].sNum[7].rPercent, nameStr3 := gUI.DiG.arrPV[7].sNum[8].strName, posVal3 := gUI.DiG.arrPV[7].sNum[8].rPosition, percentBar3 := gUI.DiG.arrPV[7].sNum[8].rPercent, nameStr4 := gUI.DiG.arrPV[7].sNum[9].strName, posVal4 := gUI.DiG.arrPV[7].sNum[9].rPosition, percentBar4 := gUI.DiG.arrPV[7].sNum[9].rPercent)
    Frame (306,181 692x156), "04"
        shows ModuleX5(extendButton := gUI.DiG.arrPV[7].sColumn[4].bExtend, retractButton := gUI.DiG.arrPV[7].sColumn[4].bRetract, stopButton := gUI.DiG.arrPV[7].sColumn[4].bStop, nameStr1 := gUI.DiG.arrPV[7].sNum[10].strName, posVal1 := gUI.DiG.arrPV[7].sNum[10].rPosition, percentBar1 := gUI.DiG.arrPV[7].sNum[10].rPercent, nameStr2 := gUI.DiG.arrPV[7].sNum[11].strName, posVal2 := gUI.DiG.arrPV[7].sNum[11].rPosition, percentBar2 := gUI.DiG.arrPV[7].sNum[11].rPercent, nameStr3 := gUI.DiG.arrPV[7].sNum[12].strName, posVal3 := gUI.DiG.arrPV[7].sNum[12].rPosition, percentBar3 := gUI.DiG.arrPV[7].sNum[12].rPercent, nameStr4 := gUI.DiG.arrPV[7].sNum[13].strName, posVal4 := gUI.DiG.arrPV[7].sNum[13].rPosition, percentBar4 := gUI.DiG.arrPV[7].sNum[13].rPercent, nameStr5 := gUI.DiG.arrPV[7].sNum[14].strName, posVal5 := gUI.DiG.arrPV[7].sNum[14].rPosition, percentBar5 := gUI.DiG.arrPV[7].sNum[14].rPercent)
    Frame (306,350 692x156), "05"
        shows ModuleX5(extendButton := gUI.DiG.arrPV[7].sColumn[5].bExtend, retractButton := gUI.DiG.arrPV[7].sColumn[5].bRetract, stopButton := gUI.DiG.arrPV[7].sColumn[5].bStop, nameStr1 := gUI.DiG.arrPV[7].sNum[15].strName, posVal1 := gUI.DiG.arrPV[7].sNum[15].rPosition, percentBar1 := gUI.DiG.arrPV[7].sNum[15].rPercent, nameStr2 := gUI.DiG.arrPV[7].sNum[16].strName, posVal2 := gUI.DiG.arrPV[7].sNum[16].rPosition, percentBar2 := gUI.DiG.arrPV[7].sNum[16].rPercent, nameStr3 := gUI.DiG.arrPV[7].sNum[17].strName, posVal3 := gUI.DiG.arrPV[7].sNum[17].rPosition, percentBar3 := gUI.DiG.arrPV[7].sNum[17].rPercent, nameStr4 := gUI.DiG.arrPV[7].sNum[18].strName, posVal4 := gUI.DiG.arrPV[7].sNum[18].rPosition, percentBar4 := gUI.DiG.arrPV[7].sNum[18].rPercent, nameStr5 := gUI.DiG.arrPV[7].sNum[19].strName, posVal5 := gUI.DiG.arrPV[7].sNum[19].rPosition, percentBar5 := gUI.DiG.arrPV[7].sNum[19].rPercent)
    Frame (0,183 292x156), "06"
        shows ModuleX2(extendButton := gUI.DiG.arrPV[7].sColumn[6].bExtend, retractButton := gUI.DiG.arrPV[7].sColumn[6].bRetract, stopButton := gUI.DiG.arrPV[7].sColumn[6].bStop, nameStr1 := gUI.DiG.arrPV[7].sNum[20].strName, posVal1 := gUI.DiG.arrPV[7].sNum[20].rPosition, percentBar1 := gUI.DiG.arrPV[7].sNum[20].rPercent, nameStr2 := gUI.DiG.arrPV[7].sNum[21].strName, posVal2 := gUI.DiG.arrPV[7].sNum[21].rPosition, percentBar2 := gUI.DiG.arrPV[7].sNum[21].rPercent)
    Frame (0,350 292x156), "07"
        shows ModuleX2(extendButton := gUI.DiG.arrPV[7].sColumn[7].bExtend, retractButton := gUI.DiG.arrPV[7].sColumn[7].bRetract, stopButton := gUI.DiG.arrPV[7].sColumn[7].bStop, nameStr1 := gUI.DiG.arrPV[7].sNum[22].strName, posVal1 := gUI.DiG.arrPV[7].sNum[22].rPosition, percentBar1 := gUI.DiG.arrPV[7].sNum[22].rPercent, nameStr2 := gUI.DiG.arrPV[7].sNum[23].strName, posVal2 := gUI.DiG.arrPV[7].sNum[23].rPosition, percentBar2 := gUI.DiG.arrPV[7].sNum[23].rPercent)
    Frame (1035,385 261x106)
        shows ModuleDTD(enable := gUI.DiG.arrPV[7].bPVD_enable, propPercent := gUI.DiG.arrPV[7].rPVDPercent)
END_VISUALIZATION

// Device/Application/display/OrigDi/Floor_Rail_67ByNum
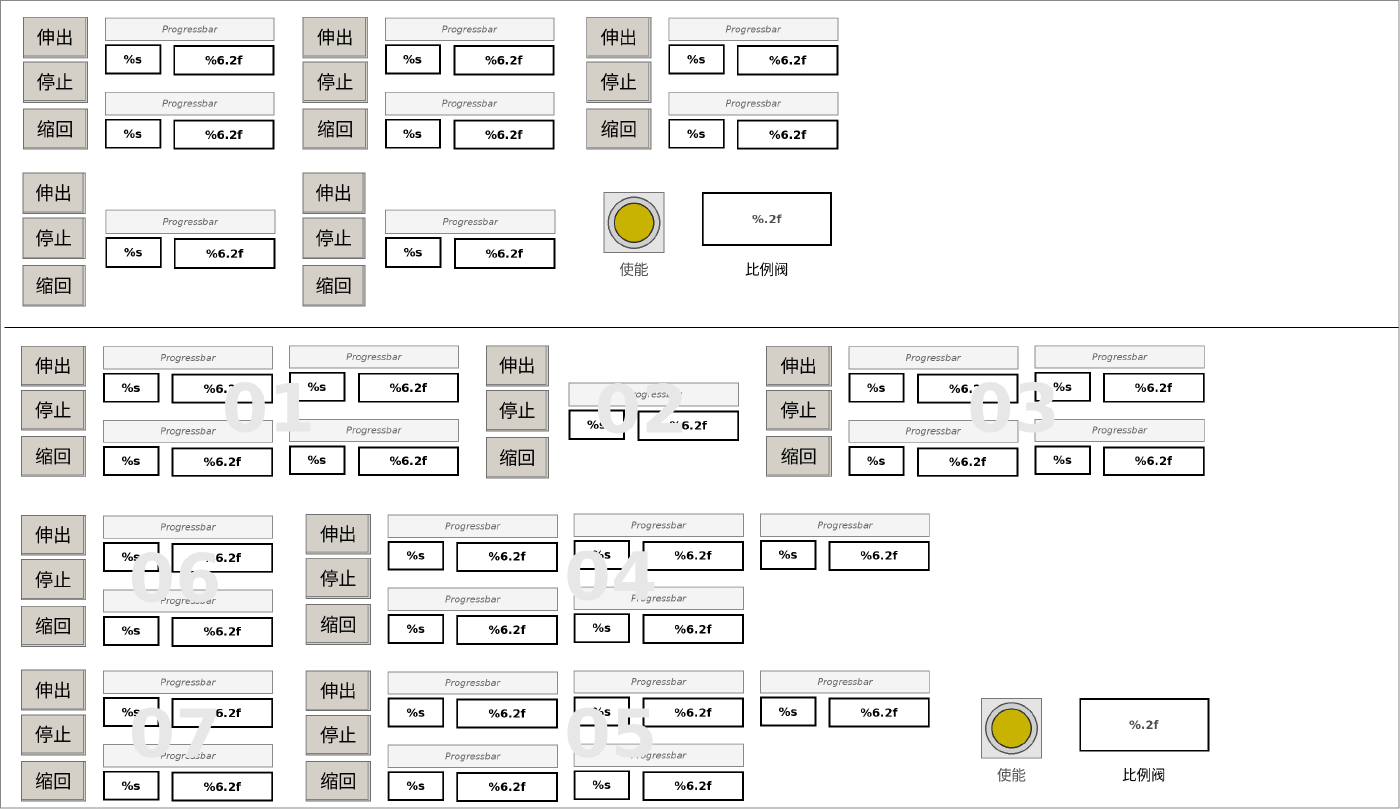
VISUALIZATION Floor_Rail_67ByNum  // 1502x868
    Frame (5,5 900x330)
        shows Floor_Rail6()
    Line (5,351) (1500,351)
    Frame (5,360 1296x506)
        shows Floor_Rail7_ByNum()
END_VISUALIZATION

// Device/Application/display/OrigDi/Floor_Rail
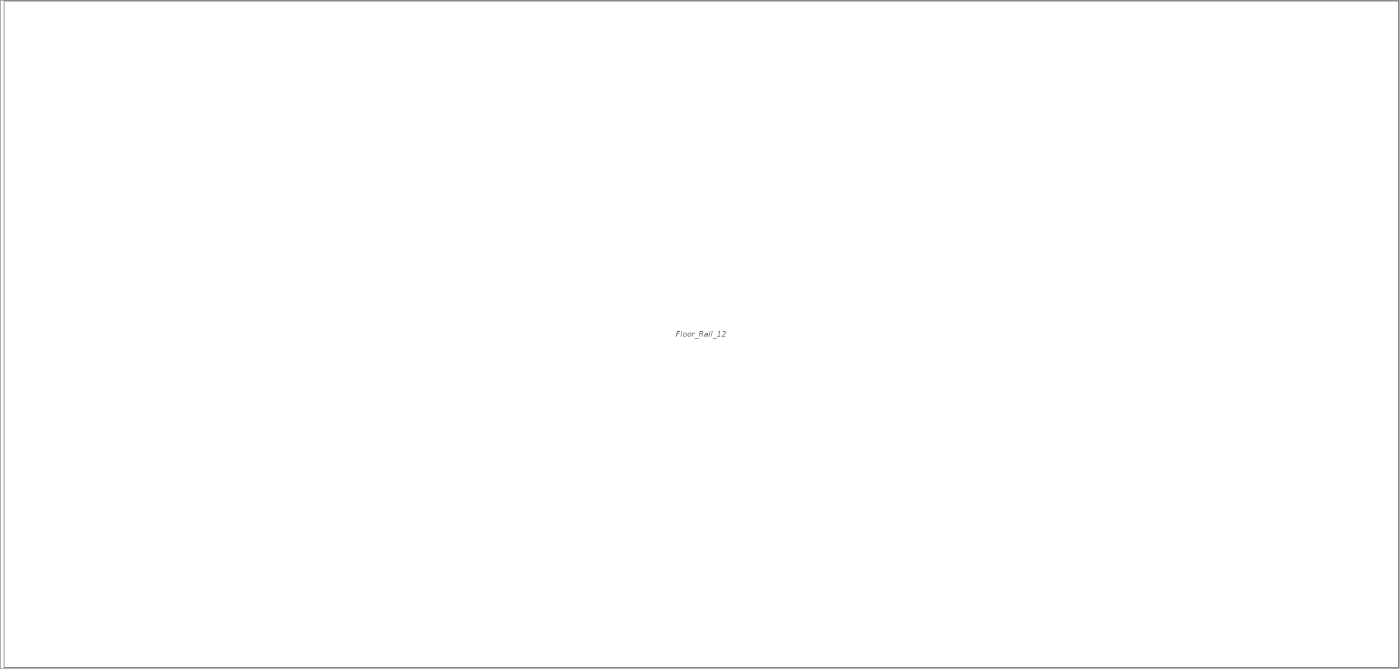
VISUALIZATION Floor_Rail  // 1847x883
    TabControl (5,1 1840x880)
        shows Floor_Rail_12()
        shows Floor_Rail_345()
        shows Floor_Rail_67ByNum()
        [0]: TabTitle=地轨1-2, ImageId=__VisualizationStyle.Element-Clock-Blue
        [1]: TabTitle=地轨3-5, ImageId=__VisualizationStyle.Element-Clock-Blue
        [2]: TabTitle=地轨6-7, ImageId=__VisualizationStyle.Element-Clock-Blue
END_VISUALIZATION

// Device/Application/display/OrigTi/Ceiling_Rail1
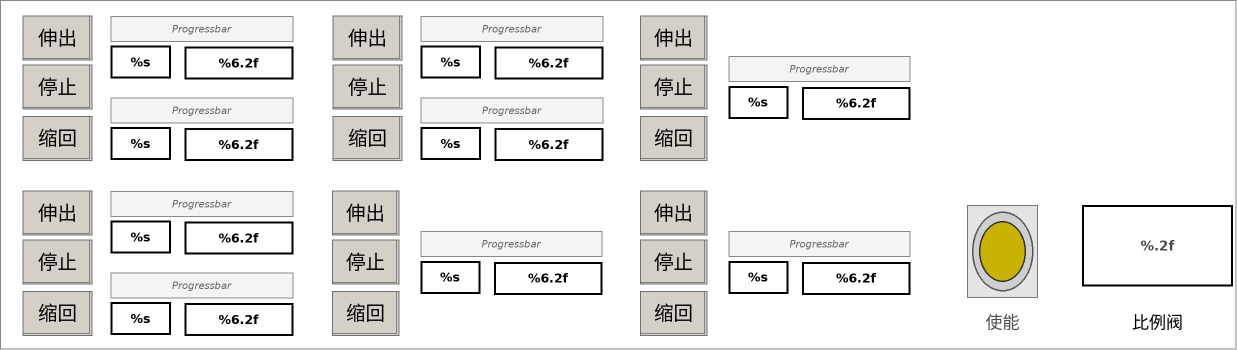
VISUALIZATION Ceiling_Rail1  // 1237x350
    Frame (5,5 292x160)
        shows ModuleX2(extendButton := gUI.TiG.arrPV[1].sColumn[1].bExtend, retractButton := gUI.TiG.arrPV[1].sColumn[1].bRetract, stopButton := gUI.TiG.arrPV[1].sColumn[1].bStop, nameStr1 := gUI.TiG.arrPV[1].sNum[1].strName, posVal1 := gUI.TiG.arrPV[1].sNum[1].rPosition, percentBar1 := gUI.TiG.arrPV[1].sNum[1].rPercent, nameStr2 := gUI.TiG.arrPV[1].sNum[2].strName, posVal2 := gUI.TiG.arrPV[1].sNum[2].rPosition, percentBar2 := gUI.TiG.arrPV[1].sNum[2].rPercent)
    Frame (315,5 292x160)
        shows ModuleX2(extendButton := gUI.TiG.arrPV[1].sColumn[2].bExtend, retractButton := gUI.TiG.arrPV[1].sColumn[2].bRetract, stopButton := gUI.TiG.arrPV[1].sColumn[2].bStop, nameStr1 := gUI.TiG.arrPV[1].sNum[3].strName, posVal1 := gUI.TiG.arrPV[1].sNum[3].rPosition, percentBar1 := gUI.TiG.arrPV[1].sNum[3].rPercent, nameStr2 := gUI.TiG.arrPV[1].sNum[4].strName, posVal2 := gUI.TiG.arrPV[1].sNum[4].rPosition, percentBar2 := gUI.TiG.arrPV[1].sNum[4].rPercent)
    Frame (5,180 292x160)
        shows ModuleX2(extendButton := gUI.TiG.arrPV[1].sColumn[4].bExtend, retractButton := gUI.TiG.arrPV[1].sColumn[4].bRetract, stopButton := gUI.TiG.arrPV[1].sColumn[4].bStop, nameStr1 := gUI.TiG.arrPV[1].sNum[6].strName, posVal1 := gUI.TiG.arrPV[1].sNum[6].rPosition, percentBar1 := gUI.TiG.arrPV[1].sNum[6].rPercent, nameStr2 := gUI.TiG.arrPV[1].sNum[7].strName, posVal2 := gUI.TiG.arrPV[1].sNum[7].rPosition, percentBar2 := gUI.TiG.arrPV[1].sNum[7].rPercent)
    Frame (952,197 283x151)
        shows ModuleDTD(enable := gUI.TiG.arrPV[1].bPVD_enable, propPercent := gUI.TiG.arrPV[1].rPVDPercent)
    Frame (623,5 291x160)
        shows ModuleX1(extendButton := gUI.TiG.arrPV[1].sColumn[3].bExtend, retractButton := gUI.TiG.arrPV[1].sColumn[3].bRetract, stopButton := gUI.TiG.arrPV[1].sColumn[3].bStop, nameStr := gUI.TiG.arrPV[1].sNum[5].strName, posVal := gUI.TiG.arrPV[1].sNum[5].rPosition, percentBar := gUI.TiG.arrPV[1].sNum[5].rPercent)
    Frame (315,180 291x160)
        shows ModuleX1(extendButton := gUI.TiG.arrPV[1].sColumn[5].bExtend, retractButton := gUI.TiG.arrPV[1].sColumn[5].bRetract, stopButton := gUI.TiG.arrPV[1].sColumn[5].bStop, nameStr := gUI.TiG.arrPV[1].sNum[8].strName, posVal := gUI.TiG.arrPV[1].sNum[8].rPosition, percentBar := gUI.TiG.arrPV[1].sNum[8].rPercent)
    Frame (623,180 291x160)
        shows ModuleX1(extendButton := gUI.TiG.arrPV[1].sColumn[6].bExtend, retractButton := gUI.TiG.arrPV[1].sColumn[6].bRetract, stopButton := gUI.TiG.arrPV[1].sColumn[6].bStop, nameStr := gUI.TiG.arrPV[1].sNum[9].strName, posVal := gUI.TiG.arrPV[1].sNum[9].rPosition, percentBar := gUI.TiG.arrPV[1].sNum[9].rPercent)
END_VISUALIZATION

// Device/Application/display/OrigDi/Floor_Rail2
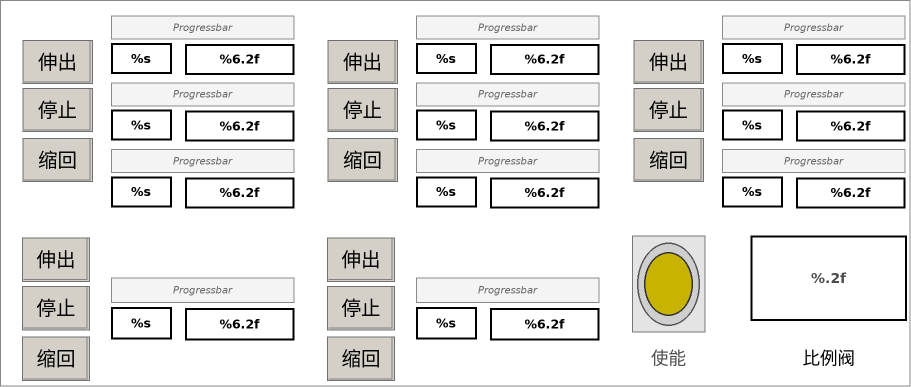
VISUALIZATION Floor_Rail2  // 911x387
    Frame (5,5 293x207)
        shows ModuleX3(extendButton := gUI.DiG.arrPV[2].sColumn[1].bExtend, retractButton := gUI.DiG.arrPV[2].sColumn[1].bRetract, stopButton := gUI.DiG.arrPV[2].sColumn[1].bStop, nameStr1 := gUI.DiG.arrPV[2].sNum[1].strName, posVal1 := gUI.DiG.arrPV[2].sNum[1].rPosition, percentBar1 := gUI.DiG.arrPV[2].sNum[1].rPercent, nameStr2 := gUI.DiG.arrPV[2].sNum[2].strName, posVal2 := gUI.DiG.arrPV[2].sNum[2].rPosition, percentBar2 := gUI.DiG.arrPV[2].sNum[2].rPercent, nameStr3 := gUI.DiG.arrPV[2].sNum[3].strName, posVal3 := gUI.DiG.arrPV[2].sNum[3].rPosition, percentBar3 := gUI.DiG.arrPV[2].sNum[3].rPercent)
    Frame (5,227 293x158)
        shows ModuleX1(extendButton := gUI.DiG.arrPV[2].sColumn[2].bExtend, retractButton := gUI.DiG.arrPV[2].sColumn[2].bRetract, stopButton := gUI.DiG.arrPV[2].sColumn[2].bStop, nameStr := gUI.DiG.arrPV[2].sNum[4].strName, posVal := gUI.DiG.arrPV[2].sNum[4].rPosition, percentBar := gUI.DiG.arrPV[2].sNum[4].rPercent)
    Frame (310,5 293x207)
        shows ModuleX3(extendButton := gUI.DiG.arrPV[2].sColumn[3].bExtend, retractButton := gUI.DiG.arrPV[2].sColumn[3].bRetract, stopButton := gUI.DiG.arrPV[2].sColumn[3].bStop, nameStr1 := gUI.DiG.arrPV[2].sNum[5].strName, posVal1 := gUI.DiG.arrPV[2].sNum[5].rPosition, percentBar1 := gUI.DiG.arrPV[2].sNum[5].rPercent, nameStr2 := gUI.DiG.arrPV[2].sNum[6].strName, posVal2 := gUI.DiG.arrPV[2].sNum[6].rPosition, percentBar2 := gUI.DiG.arrPV[2].sNum[6].rPercent, nameStr3 := gUI.DiG.arrPV[2].sNum[7].strName, posVal3 := gUI.DiG.arrPV[2].sNum[7].rPosition, percentBar3 := gUI.DiG.arrPV[2].sNum[7].rPercent)
    Frame (310,227 293x158)
        shows ModuleX1(extendButton := gUI.DiG.arrPV[2].sColumn[4].bExtend, retractButton := gUI.DiG.arrPV[2].sColumn[4].bRetract, stopButton := gUI.DiG.arrPV[2].sColumn[4].bStop, nameStr := gUI.DiG.arrPV[2].sNum[8].strName, posVal := gUI.DiG.arrPV[2].sNum[8].rPosition, percentBar := gUI.DiG.arrPV[2].sNum[8].rPercent)
    Frame (616,5 293x207)
        shows ModuleX3(extendButton := gUI.DiG.arrPV[2].sColumn[5].bExtend, retractButton := gUI.DiG.arrPV[2].sColumn[5].bRetract, stopButton := gUI.DiG.arrPV[2].sColumn[5].bStop, nameStr1 := gUI.DiG.arrPV[2].sNum[9].strName, posVal1 := gUI.DiG.arrPV[2].sNum[9].rPosition, percentBar1 := gUI.DiG.arrPV[2].sNum[9].rPercent, nameStr2 := gUI.DiG.arrPV[2].sNum[10].strName, posVal2 := gUI.DiG.arrPV[2].sNum[10].rPosition, percentBar2 := gUI.DiG.arrPV[2].sNum[10].rPercent, nameStr3 := gUI.DiG.arrPV[2].sNum[11].strName, posVal3 := gUI.DiG.arrPV[2].sNum[11].rPosition, percentBar3 := gUI.DiG.arrPV[2].sNum[11].rPercent)
    Frame (616,227 293x158)
        shows ModuleDTD(enable := gUI.TiG.arrPV[2].bPVD_enable, propPercent := gUI.TiG.arrPV[2].rPVDPercent)
END_VISUALIZATION

// Device/Application/display/OrigTi/Ceiling_Rail_345
